(* Logix 5000 project; controller LeakTestAuto vendor 1 type 14 code 226 rev 37.11; software revision 37.01; part 3 of 13 *)
(* tags used below, declared in another part *)
   iarsiInputFromDTE : SINT[496];   // Input array from DTE to PLC
   iiInputStartAdd : INT;   // It is the start of the DTE102:I from which the data has to be read depending upon the channel is being used by the user
   oarsiOutputToDTE : SINT[496];   // Output array from PLC to DTE
   iLoopHandlerVar1 : INT;   // Local tag - Loop Handler variable 1
   iArraySize : INT;
   scDTE102_Handling : DTE102_CmdModule;
   iStateMachine_RWH_CMD : INT;   // Local tag - State machine handling variable for AOI logic
(* RWH_CMD, continued *)

ROUTINE Prescan   (* structured text *)
// Intialisation routine
   	(*Intialise*)
   
   	scDTE102_Handling.ActivateCommand.AO	:= 0;
   	scDTE102_Handling.ActivateCommand.WR	:= 0;
   	scDTE102_Handling.ActivateCommand.RD	:= 0;
   	scDTE102_Handling.ActivateCommand.UR	:= 0;
   	scDTE102_Handling.ActivateCommand.ER	:= 0;
   	scDTE102_Handling.ActivateCommand.DR	:= 0;
   	scDTE102_Handling.ActivateCommand.CM	:= 0;
   	scDTE102_Handling.ActivateCommand.TR	:= (iarsiInputFromDTE[iiInputStartAdd+1].0);
   
   	SIZE(oarsiOutputToDTE,0,iArraySize);
   	FOR iLoopHandlerVar1 :=0 TO iArraySize BY 1 DO;
           oarsiOutputToDTE[iLoopHandlerVar1] := 0;
       END_FOR;
   
   	iStateMachine_RWH_CMD := 25999;
   
END_ROUTINE
END_ADD_ON_INSTRUCTION

ADD_ON_INSTRUCTION SINT_TO_INT   (* revision 1.0 *)
// Converts the negative values of SINT variable to positive values and stores it to a INT variable.
// -128 to -1 = 128 to 255
// 0 to 127 = 0 to 127
// So -128 to 127 to 0 to 255
VAR_INPUT
   iSINT_var : SINT; {required}
END_VAR
VAR_OUTPUT
   oINT_var : INT; {visible}
END_VAR

ROUTINE Logic   (* structured text *)
   IF(iSINT_var<0)THEN
   	oINT_var := 256 + iSINT_var;
   ELSE
   	oINT_var := iSINT_var;
   END_IF;
END_ROUTINE
END_ADD_ON_INSTRUCTION

VAR_GLOBAL   (* controller tags *)
   AOI_IOCounter : AOI_IOCounter;
   ConveyorPurgeCounter : DINT;   // Outfeed Coveyor Purge Counter
   DateString : String20 := '01/14/1998';
   DateTimeString : String20 := '01/14/1998 03:13:45';
   Delay_TMR : TIMER[11] := ([0].PRE := 500, [1].PRE := 500, [3].PRE := 1000, [10].PRE := 100);   // Delay Timers
   HMI_ClearProcessFaultCounts_PB : BOOL;
   HMI_PurgeCycleSP : DINT := 20;   // HMI Purge Cycles Setpoint
   I_OP220_N3_CONVEYOR_CLEAT : ALIAS FOR Local:3:I.Pt13.Data;
   I_OP220_N3_CONVEYOR_LOAD : ALIAS FOR Local:3:I.Pt12.Data;
   I_OP220_N3_CONVEYOR_UNLOAD : ALIAS FOR Local:3:I.Pt14.Data;
   I_OP220_N3_CTS_AIR_OK : ALIAS FOR Local:3:I.Pt08.Data;
   I_OP220_N3_DUT_PRE_NEST_0 : ALIAS FOR Local:3:I.Pt00.Data;
   I_OP220_N3_DUT_PRE_NEST_1 : ALIAS FOR Local:3:I.Pt01.Data;
   I_OP220_N3_DUT_PRE_NEST_2 : ALIAS FOR Local:3:I.Pt02.Data;
   I_OP220_N3_MAIN_AIR_OK : ALIAS FOR Local:3:I.Pt07.Data;
   I_OP220_N3_NEST1_EXTEND : ALIAS FOR Local:3:I.Pt04.Data;
   I_OP220_N3_NEST1_HOME : ALIAS FOR Local:3:I.Pt03.Data;
   I_OP220_N3_NEST2_EXTEND : ALIAS FOR Local:3:I.Pt06.Data;
   I_OP220_N3_NEST2_HOME : ALIAS FOR Local:3:I.Pt05.Data;
   I_OP220_N3_REJECT_BIN_OK : ALIAS FOR Local:3:I.Pt09.Data;
   I_OP220_N3_REJECT_CHUTE_PART : ALIAS FOR Local:3:I.Pt10.Data;
   I_OP220_N4_AC_SURGE_OK : ALIAS FOR Local:4:I.Pt00.Data;
   I_OP220_N4_CONVEYOR_ALARM_OK : ALIAS FOR Local:4:I.Pt03.Data;
   I_OP220_N4_CONVEYOR_SPEED : ALIAS FOR Local:4:I.Pt02.Data;
   I_OP220_N4_DC_OK : ALIAS FOR Local:4:I.Pt01.Data;
   I_OP220_N4_DC_OK_PS2 : ALIAS FOR Local:4:I.Pt04.Data;
   Ignition_Bypass : BOOL := 1;
   Ignition_DataReady : BOOL;
   Ignition_DataReceived : BOOL;
   IOCounterHasRef : BOOL := 1;
   IOCounterLastData : INT[8] := ([0] := 13997, [1] := 27, [2] := -31920);
   IOLabels : STRING[128] := ([0] := 'SI_OP220_N1_LASER_AREA_NC12', [1] := 'SI_OP220_N1_LASER_GUARD_NC12', [3] := 'SI_OP220_N1_SSR_12', [4] := 'SI_OP220_N1_CTRL_VLAVE_NC1', [8] := 'SO_OP220_N2_SSR_1', [9] := 'SO_OP220_N2_SSR_2', [16] := 'I_OP220_N3_DUT_PRE_NEST_0', [17] := 'I_OP220_N3_DUT_PRE_NEST_1', [18] := 'I_OP220_N3_DUT_PRE_NEST_2', [19] := 'I_OP220_N3_NEST1_HOME', [20] := 'I_OP220_N3_NEST1_EXTEND', [21] := 'I_OP220_N3_NEST2_HOME', [22] := 'I_OP220_N3_NEST2_EXTEND', [23] := 'I_OP220_N3_MAIN_AIR_OK', [25] := 'I_OP220_N3_REJECT_BIN_OK', [26] := 'I_OP220_N3_REJECT_CHUTE_PART', [28] := 'I_OP220_N3_CONVEYOR_LOAD', [29] := 'I_OP220_N3_CONVEYOR_CLEAT', [30] := 'I_OP220_N3_CONVEYOR_UNLOAD', [32] := 'I_OP220_N4_AC_SURGE_OK', [33] := 'I_OP220_N4_DC_OK', [34] := 'I_OP220_N4_CONVEYOR_SPEED', [35] := 'I_OP220_N4_CONVEYOR_ALARM_OK', [36] := 'I_OP220_N4_DC_OK_PS2', [48] := 'O_OP220_N5_EN_LT_GN', [49] := 'O_OP220_N5_EN_LT_YE', [50] := 'O_OP220_N5_EN_LT_RD', [51] := 'O_OP220_N5_EN_LT_BU', [52] := 'O_OP220_N5_EN_MAIN_AIR', [53] := 'O_OP220_N5_EN_NEST1_EXT', [54] := 'O_OP220_N5_EN_NEST1_HOME', [55] := 'O_OP220_N5_EN_NEST2_EXT', [56] := 'O_OP220_N5_EN_NEST2_HOME', [57] := 'O_OP220_N5_EN_ROBOT_LATCHOFF', [58] := 'O_OP220_N5_EN_CONV_ALM_RST', [59] := 'O_OP220_N5_CONV_REV', [60] := 'O_OP220_N5_CONV_FWD', [62] := 'O_OP220_N5_EN_GRIPPER_GRIP', [63] := 'O_OP220_N5_EN_GRIPPER_UNGRIP');
   IOResetArray : INT[8];
   IOTriggerCounts : UDINT[128] := ([0] := 204475, [1] := 372996, [2] := 290087, [3] := 284, [4] := 293, [5] := 289, [6] := 294, [7] := 60, [8] := 522, [9] := 268, [10] := 461, [11] := 1169, [12] := 501, [13] := 259, [14] := 218085, [16] := 969915, [17] := 969727, [18] := 63, [19] := 1025, [21] := 84232, [22] := 84239, [23] := 72816, [24] := 72798, [25] := 504, [26] := 4412, [28] := 201969, [29] := 3, [30] := 359118, [31] := 359118);
   James_Dint : DINT := 31;   // James Test Word
   LastPLCEdit : String20 := '01/14/1998 03:11:29';
   LastPLCEditHistory : String20[20] := ([0] := '01/14/1998 03:11:29', [1] := '01/14/1998 02:38:23', [2] := '01/14/1998 02:28:45', [3] := '01/14/1998 02:24:53', [4] := '01/11/1998 11:02:53', [5] := '01/11/1998 10:59:23', [6] := '01/11/1998 10:58:09', [7] := '01/11/1998 10:55:51', [8] := '01/11/1998 05:50:18', [9] := '01/11/1998 05:46:44', [10] := '01/11/1998 05:46:03', [11] := '01/11/1998 05:24:08', [12] := '01/11/1998 05:15:43', [13] := '01/11/1998 04:51:18', [14] := '01/11/1998 04:33:38', [15] := '01/11/1998 03:28:20', [16] := '01/10/1998 12:07:04', [17] := '01/10/1998 12:06:39', [18] := '01/10/1998 12:05:41', [19] := '01/10/1998 11:56:52');
   NoData : AB:5000_DI16:I:0;
   null : STRING;
   O_OP220_N5_CONV_FWD : ALIAS FOR Local:5:O.Pt12.Data;
   O_OP220_N5_CONV_REV : ALIAS FOR Local:5:O.Pt11.Data;
   O_OP220_N5_EN_CONV_ALM_RST : ALIAS FOR Local:5:O.Pt10.Data;
   O_OP220_N5_EN_GRIPPER_GRIP : ALIAS FOR Local:5:O.Pt14.Data;
   O_OP220_N5_EN_GRIPPER_UNGRIP : ALIAS FOR Local:5:O.Pt15.Data;
   O_OP220_N5_EN_LT_BU : ALIAS FOR Local:5:O.Pt03.Data;
   O_OP220_N5_EN_LT_GN : ALIAS FOR Local:5:O.Pt00.Data;
   O_OP220_N5_EN_LT_RD : ALIAS FOR Local:5:O.Pt02.Data;
   O_OP220_N5_EN_LT_YE : ALIAS FOR Local:5:O.Pt01.Data;
   O_OP220_N5_EN_MAIN_AIR : ALIAS FOR Local:5:O.Pt04.Data;
   O_OP220_N5_EN_NEST1_EXT : ALIAS FOR Local:5:O.Pt05.Data;
   O_OP220_N5_EN_NEST1_HOME : ALIAS FOR Local:5:O.Pt06.Data;
   O_OP220_N5_EN_NEST2_EXT : ALIAS FOR Local:5:O.Pt07.Data;
   O_OP220_N5_EN_NEST2_HOME : ALIAS FOR Local:5:O.Pt08.Data;
   O_OP220_N5_EN_ROBOT_LATCHOFF : ALIAS FOR Local:5:O.Pt09.Data;
   Oneshot : DINT;   // Oneshots
   OP220_ConsumedFromMain : DINT[50] := ([0] := 2, [1] := 2);
   OP220_ConsumedFromMain_PurgeModeEn : BOOL;
   OP220_ConsumedFromMain_RobotPickupSafe : BOOL := 1;
   OP220_EStop_OK : BOOL := 1;
   OP220_EStopTest_DCS : DCI_STOP := (ChannelA := 1, ChannelB := 1, InputStatus := 1, RestartType := 1, ColdStartType := 1, DiscrepancyTime := 250, O1 := 1);
   OP220_Power : BOOL := 1;
   OP220_ProducedForMain : DINT[50] := ([0] := 3); {produced}
   PLC : AOI_PLC := (AlwaysOn := 1, FlasherSlow := 1, SlowFlashTime := 2000, MediumFlashTime := 1000, FastFlashTime := 500, Year := 1998, Day := 14, Month := 1, Hour := 3, Minute := 13, Second := 45, MicroSecond := 714855, DOY := 14, SetTimePB := 1);
   Produced_SetTime : udt_Produced_SetTime := (SetTime[0] := 2020, SetTime[1] := 5, SetTime[2] := 21, SetTime[3] := 15, SetTime[4] := 59, SetTime[5] := 15); {produced}
   Purge_Count_DN : BOOL;   // Purge Counter Completed
   ShiftChange : BOOL;
   ShiftNumber : SINT := 2;
   SI_OP220_N1_CTRL_VLAVE_NC1 : ALIAS FOR Local:1:I.Pt04.Data;
   SI_OP220_N1_LASER_AREA_NC12 : ALIAS FOR Local:1:I.Pt00.Data;
   SI_OP220_N1_LASER_GUARD_NC12 : ALIAS FOR Local:1:I.Pt01.Data;
   SI_OP220_N1_SSR_12 : ALIAS FOR Local:1:I.Pt03.Data;
   SO_OP220_N2_SSR_1 : ALIAS FOR Local:2:O.Pt00.Data;
   SO_OP220_N2_SSR_2 : ALIAS FOR Local:2:O.Pt01.Data;
   ST1_Ignition_DataReady : BOOL;
   ST1_Ignition_DataReady_Setup : BOOL;
   ST1_Ignition_DataReceived : BOOL;
   ST1_Ignition_SerialNum : STRING;
   ST1_Ignition_Status : DINT := -10;
   ST2_Ignition_DataReady : BOOL;
   ST2_Ignition_DataReady_Setup : BOOL;
   ST2_Ignition_DataReceived : BOOL;
   ST2_Ignition_SerialNum : STRING;
   ST2_Ignition_Status : DINT := -10;
   TimeString : String20 := '03:13:45';
   TON_PLC_BootUp : TIMER := (PRE := 10000);
END_VAR

PROGRAM MainProgram   (* main routine MainRoutine *)
VAR
   AOI_Barcode_Comms : AOI_CommStatus := (Cmd := 1, stsRunning := 1, stsFaultCode := 272);
   AOI_CapActuators_Seq : AOI_Sequencer_x64 := (inpNextStepInterlock := 1);
   AOI_CapCTS_Seq : AOI_Sequencer_x64 := (inpNextStepInterlock := 1);
   AOI_CapCylinders_Seq : AOI_Sequencer_x64 := (inpNextStepInterlock := 1);
   AOI_CapFail_Seq : AOI_Sequencer_x64 := (inpNextStepInterlock := 1);
   AOI_CapPass_Seq : AOI_Sequencer_x64 := (inpNextStepInterlock := 1);
   AOI_CapRobot_Seq : AOI_Sequencer_x64 := (inpNextStepInterlock := 1);
   AOI_CapShuffle_Seq : AOI_Sequencer_x64 := (inpNextStepInterlock := 1);
   AOI_Conveyor_Seq : AOI_Sequencer_x64 := (inpNextStepInterlock := 1);
   AOI_CTS1 : AOI_CTS_INSTRUMENT := (Change_Program_Number := 3, Current_Program_Number := 3, Instrument_Ready := 1, Program_Accept := 1, Last_Result_Unique_ID := 9525, Last_Result_Channel_Number := 1, Last_Result_Progam_Number := 3, Last_Result_Evaluation_Code := 1, Last_Result_Year := 26, Last_Result_Month := 9, Last_Result_Date := 28, Last_Result_Hour := 11, Last_Result_Minute := 13, Last_Result_Second := 13, UID_of_Desired_Results := 9478, Include_Detailed_Results := 1, Results_Ready := 1, UID_Time := 1300, Ready := 1);
   AOI_CTS1_Comms : AOI_CommStatus := (Cmd := 1, stsRunning := 1, stsFaultCode := 272);
   AOI_CTS1_Seq : AOI_Sequencer_x64 := (inpNextStepInterlock := 1);
   AOI_CTS2 : AOI_CTS_INSTRUMENT := (Change_Program_Number := 3, Current_Program_Number := 3, Instrument_Ready := 1, Program_Accept := 1, Last_Result_Unique_ID := 10924, Last_Result_Channel_Number := 1, Last_Result_Progam_Number := 3, Last_Result_Evaluation_Code := 1, Last_Result_Year := 26, Last_Result_Month := 9, Last_Result_Date := 28, Last_Result_Hour := 11, Last_Result_Second := 7, UID_of_Desired_Results := 10592, Include_Detailed_Results := 1, Results_Ready := 1, UID_Time := 1300, Ready := 1);
   AOI_CTS2_Comms : AOI_CommStatus := (Cmd := 1, stsRunning := 1, stsFaultCode := 272);
   AOI_CTS2_Seq : AOI_Sequencer_x64 := (inpNextStepInterlock := 1);
   AOI_GetShift : AOI_GetShift := (PLCHour := 3, ShiftNumber := 2);
   AOI_OP220_HomingSeq : AOI_Sequencer_x64;
   AOI_OP220_Seq : AOI_Sequencer_x64 := (inpNextStepInterlock := 1);
   AOI_RFID_Comms : AOI_CommStatus := (Cmd := 1, stsRunning := 1, stsFaultCode := 516);
   AOI_RFID_LoadingNest_Comms : AOI_CommStatus := (Cmd := 1, stsRunning := 1, stsFaultCode := 272);
   AOI_Robot_Comms : AOI_CommStatus := (Cmd := 1, stsRunning := 1, stsFaultCode := 272);
   AOI_RobotPos : AOI_RobotPositions := (Barcode := 1, TestingNest1 := 2, TestingNest2 := 3, PassChute := 4, FailChute := 5);
   AOI_SeqSteps : AOI_StandardSeqSteps := (Start := 1000, ResultProcessing := 8000, Complete := 9000);
   AOI_SRX100 : AOI_KeyenceBarcode := (ReadSuccess := 1);
   Barcode_ResultData : STR_Barcode := '260911463C';
   BarcodeBypass : BOOL;
   BarcodeInputs : udt_KeyenceScannerInputs := (READY := 1, ResultDataReadyCount := 25, ResultDataUpdateCount := 25, MasterTriggerCount := 25, ResultDataSize := 10, ResultData[0] := 50, ResultData[1] := 54, ResultData[2] := 48, ResultData[3] := 51, ResultData[4] := 56, ResultData[5] := 48, ResultData[6] := 56, ResultData[7] := 48, ResultData[8] := 57, ResultData[9] := 67);
   BarcodeOutputs : udt_KeyenceScannerOutputs;
   BarcodeScanner : udt_OutputStructure := (IL := 1);
   CapActuators_BarcodeBad : COUNTER := (PRE := 999999999, CU := 1);
   CapActuators_BarcodeGood : COUNTER := (PRE := 999999999, ACC := 111, CU := 1);
   CapActuators_CTS1Bad : COUNTER := (PRE := 999999999, CU := 1);
   CapActuators_CTS1Good : COUNTER := (PRE := 999999999, ACC := 10, CU := 1);
   CapActuators_CTS2Bad : COUNTER := (PRE := 999999999, CU := 1);
   CapActuators_CTS2Good : COUNTER := (PRE := 999999999, ACC := 3, CU := 1);
   CapActuators_Nest1HasPart : BOOL := 1;
   CapActuators_Nest2HasPart : BOOL;
   CapActuators_Seq : udt_SequenceStructure_X64 := (ONS := -7937, CurrentCycleTime := 409000.0, StepTimer.PRE := 999999999, CycleTimer.PRE := 999999999);
   CapCTS_CTS1Bad : COUNTER := (PRE := 999999999, ACC := 356, CU := 1);
   CapCTS_CTS1Good : COUNTER := (PRE := 999999999, ACC := 2730, CU := 1);
   CapCTS_CTS2Bad : COUNTER := (PRE := 999999999, ACC := 1, CU := 1);
   CapCTS_CTS2Good : COUNTER := (PRE := 999999999, ACC := 3085, CU := 1);
   CapCTS_Nest1HasPart : BOOL := 1;
   CapCTS_Nest2HasPart : BOOL := 1;
   CapCTS_Seq : udt_SequenceStructure_X64 := (ONS := -8132, StepHistory[0] := 2000, StepHistory[1] := 2010, StepHistory[2] := 2000, StepHistory[3] := 2010, StepHistory[4] := 2000, StepHistory[5] := 2010, StepHistory[6] := 2000, StepHistory[7] := 2010, StepHistory[8] := 2000, StepHistory[9] := 2010, StepHistory[10] := 2000, StepHistory[11] := 2010, StepHistory[12] := 2000, StepHistory[13] := 2010, StepHistory[14] := 2000, StepHistory[15] := 2010, StepHistory[16] := 2000, StepHistory[17] := 2010, StepHistory[18] := 2000, StepHistory[19] := 2010, StepHistory[20] := 2000, StepHistory[21] := 2010, StepHistory[22] := 2000, StepHistory[23] := 2010, StepHistory[24] := 2000, StepHistory[25] := 2010, StepHistory[26] := 2000, StepHistory[27] := 2010, StepHistory[28] := 2000, StepHistory[29] := 2010, StepHistory[30] := 2000, StepHistory[31] := 2010, StepHistory[32] := 2000, StepHistory[33] := 2010, StepHistory[34] := 2000, StepHistory[35] := 2010, StepHistory[36] := 2000, StepHistory[37] := 2010, StepHistory[38] := 2000, StepHistory[39] := 2010, StepHistory[40] := 2000, StepHistory[41] := 2010, StepHistory[42] := 2000, StepHistory[43] := 2010, StepHistory[44] := 2000, StepHistory[45] := 2010, StepHistory[46] := 2000, StepHistory[47] := 2010, StepHistory[48] := 2000, StepHistory[49] := 2010, StepHistory[50] := 2000, StepHistory[51] := 2010, StepHistory[52] := 2000, StepHistory[53] := 2010, StepHistory[54] := 2000, StepHistory[55] := 2010, StepHistory[56] := 2000, StepHistory[57] := 2010, StepHistory[58] := 2000,
        StepHistory[59] := 2010, StepHistory[60] := 2000, StepHistory[61] := 2010, StepHistory[62] := 2000, StepHistory[63] := 2010, CurrentCycleTime := 66060.766, CurrentStepCycleTime := 387.139, StepTimeHistory[0] := 0.035, StepTimeHistory[1] := 21.3, StepTimeHistory[2] := 0.04, StepTimeHistory[3] := 21.295, StepTimeHistory[4] := 0.035, StepTimeHistory[5] := 21.266, StepTimeHistory[6] := 0.034, StepTimeHistory[7] := 21.271, StepTimeHistory[8] := 0.033, StepTimeHistory[9] := 21.285, StepTimeHistory[10] := 0.041, StepTimeHistory[11] := 21.294, StepTimeHistory[12] := 0.052, StepTimeHistory[13] := 21.304, StepTimeHistory[14] := 0.035, StepTimeHistory[15] := 21.297, StepTimeHistory[16] := 0.036, StepTimeHistory[17] := 21.266, StepTimeHistory[18] := 0.039, StepTimeHistory[19] := 21.292, StepTimeHistory[20] := 0.04, StepTimeHistory[21] := 21.273, StepTimeHistory[22] := 0.035, StepTimeHistory[23] := 21.271, StepTimeHistory[24] := 0.051, StepTimeHistory[25] := 21.29, StepTimeHistory[26] := 0.036, StepTimeHistory[27] := 21.274, StepTimeHistory[28] := 0.041, StepTimeHistory[29] := 21.289, StepTimeHistory[30] := 0.036, StepTimeHistory[31] := 21.285, StepTimeHistory[32] := 0.039, StepTimeHistory[33] := 21.296, StepTimeHistory[34] := 0.05, StepTimeHistory[35] := 21.273, StepTimeHistory[36] := 0.057, StepTimeHistory[37] := 21.274, StepTimeHistory[38] := 0.034, StepTimeHistory[39] := 21.285, StepTimeHistory[40] := 0.05, StepTimeHistory[41] := 21.27, StepTimeHistory[42] := 0.036, StepTimeHistory[43] := 21.29, StepTimeHistory[44] := 0.035, StepTimeHistory[45] := 21.309, StepTimeHistory[46] := 0.051, StepTimeHistory[47] := 21.274, StepTimeHistory[48] := 0.037, StepTimeHistory[49] := 21.315, StepTimeHistory[50] := 0.044, StepTimeHistory[51] := 21.296, StepTimeHistory[52] := 0.035,
        StepTimeHistory[53] := 21.271, StepTimeHistory[54] := 0.034, StepTimeHistory[55] := 21.289, StepTimeHistory[56] := 0.045, StepTimeHistory[57] := 21.29, StepTimeHistory[58] := 0.034, StepTimeHistory[59] := 21.296, StepTimeHistory[60] := 0.035, StepTimeHistory[61] := 21.293, StepTimeHistory[62] := 0.069, StepTimeHistory[63] := 21.691, StepTimer.PRE := 999999999, CycleTimer.PRE := 999999999);
   CapCylinders_Seq : udt_SequenceStructure_X64 := (ONS := -8192);
   CapFail_Seq : udt_SequenceStructure_X64 := (ONS := -8192);
   CapPass_Seq : udt_SequenceStructure_X64 := (ONS := -8191);
   CapRobot_IsNest : BOOL;
   CapRobot_Seq : udt_SequenceStructure_X64 := (ONS := -8191, StepHistory[0] := 2040, StepHistory[1] := 2050, StepHistory[2] := 2060, StepHistory[3] := 2070, StepHistory[4] := 2000, StepHistory[5] := 2010, StepHistory[6] := 2020, StepHistory[7] := 2030, StepHistory[8] := 2050, StepHistory[9] := 2060, StepHistory[10] := 2070, StepHistory[11] := 2000, StepHistory[12] := 2010, StepHistory[13] := 2020, StepHistory[14] := 2030, StepHistory[15] := 2050, StepHistory[16] := 2060, StepHistory[17] := 2070, StepHistory[18] := 2000, StepHistory[19] := 2010, StepHistory[20] := 2020, StepHistory[21] := 2030, StepHistory[22] := 2040, StepHistory[23] := 2050, StepHistory[24] := 2060, StepHistory[25] := 2070, StepHistory[26] := 2000, StepHistory[27] := 2010, StepHistory[28] := 2020, StepHistory[29] := 2030, StepHistory[30] := 2040, StepHistory[31] := 2050, StepHistory[32] := 2060, StepHistory[33] := 2070, StepHistory[34] := 2000, StepHistory[35] := 2010, StepHistory[36] := 2020, StepHistory[37] := 2030, StepHistory[38] := 2050, StepHistory[39] := 2060, StepHistory[40] := 2070, StepHistory[41] := 2000, StepHistory[42] := 2010, StepHistory[43] := 2020, StepHistory[45] := 1000, StepHistory[46] := 2000, StepHistory[47] := 2010, StepHistory[48] := 2020, StepHistory[49] := 2030, StepHistory[50] := 2050, StepHistory[51] := 2060, StepHistory[52] := 2070, StepHistory[53] := 2000, StepHistory[54] := 2010, StepHistory[55] := 2020, StepHistory[56] := 2030, StepHistory[57] := 2040, StepHistory[58] := 2050, StepHistory[59] := 2060,
        StepHistory[60] := 2070, StepHistory[61] := 2000, StepHistory[62] := 2010, StepHistory[63] := 2020, CurrentCycleTime := 15.469, CurrentStepCycleTime := 4.281, StepTimeHistory[0] := 0.099, StepTimeHistory[1] := 0.039, StepTimeHistory[2] := 1.559, StepTimeHistory[3] := 1.559, StepTimeHistory[4] := 1.559, StepTimeHistory[5] := 0.097, StepTimeHistory[6] := 0.029, StepTimeHistory[7] := 1.398, StepTimeHistory[8] := 0.038, StepTimeHistory[9] := 1.468, StepTimeHistory[10] := 1.468, StepTimeHistory[11] := 1.468, StepTimeHistory[12] := 0.088, StepTimeHistory[13] := 0.028, StepTimeHistory[14] := 1.279, StepTimeHistory[15] := 0.039, StepTimeHistory[16] := 1.399, StepTimeHistory[17] := 1.399, StepTimeHistory[18] := 0.028, StepTimeHistory[19] := 0.769, StepTimeHistory[20] := 0.029, StepTimeHistory[21] := 0.758, StepTimeHistory[22] := 0.009, StepTimeHistory[23] := 0.039, StepTimeHistory[24] := 0.66, StepTimeHistory[25] := 0.66, StepTimeHistory[26] := 0.66, StepTimeHistory[27] := 0.66, StepTimeHistory[28] := 0.037, StepTimeHistory[29] := 1.209, StepTimeHistory[30] := 0.099, StepTimeHistory[31] := 0.028, StepTimeHistory[32] := 1.049, StepTimeHistory[33] := 1.049, StepTimeHistory[34] := 1.049, StepTimeHistory[35] := 1.049, StepTimeHistory[36] := 0.036, StepTimeHistory[37] := 0.898, StepTimeHistory[38] := 0.038, StepTimeHistory[39] := 0.849, StepTimeHistory[40] := 0.849, StepTimeHistory[41] := 0.849, StepTimeHistory[42] := 0.849, StepTimeHistory[43] := 0.026, StepTimeHistory[44] := 0.264, StepTimeHistory[45] := 0.264, StepTimeHistory[46] := 0.066, StepTimeHistory[47] := 1.64, StepTimeHistory[48] := 0.059, StepTimeHistory[49] := 1.569, StepTimeHistory[50] := 0.049, StepTimeHistory[51] := 1.65, StepTimeHistory[52] := 1.65, StepTimeHistory[53] := 1.65,
        StepTimeHistory[54] := 0.078, StepTimeHistory[55] := 0.058, StepTimeHistory[56] := 2.87, StepTimeHistory[57] := 0.069, StepTimeHistory[58] := 0.07, StepTimeHistory[59] := 2.87, StepTimeHistory[60] := 2.87, StepTimeHistory[61] := 2.87, StepTimeHistory[62] := 0.067, StepTimeHistory[63] := 0.06, StepTimer.PRE := 999999999, CycleTimer.PRE := 999999999);
   CapRobot_StartPos : DINT;
   CapRobot_TargetPos : DINT := 3;
   CapShuffle_CTS1Bad : COUNTER := (PRE := 999999999, ACC := 2, CU := 1);
   CapShuffle_CTS1Good : COUNTER := (PRE := 999999999, CU := 1);
   CapShuffle_CTS2Bad : COUNTER := (PRE := 999999999, CU := 1);
   CapShuffle_CTS2Good : COUNTER := (PRE := 999999999, ACC := 1, CU := 1);
   CapShuffle_Seq : udt_SequenceStructure_X64 := (ONS := -8161, StepHistory[0] := 5610, StepHistory[1] := 5620, StepHistory[2] := 5630, StepHistory[3] := 5640, StepHistory[4] := 5650, StepHistory[5] := 4000, StepHistory[6] := 4010, StepHistory[9] := 1000, StepHistory[10] := 3000, StepHistory[11] := 3010, StepHistory[12] := 3020, StepHistory[15] := 1000, StepHistory[16] := 3000, StepHistory[17] := 3010, StepHistory[18] := 3020, StepHistory[20] := 1000, StepHistory[21] := 3000, StepHistory[22] := 3010, StepHistory[23] := 3020, StepHistory[25] := 1000, StepHistory[26] := 3000, StepHistory[27] := 3010, StepHistory[28] := 3020, StepHistory[29] := 3030, StepHistory[30] := 3020, StepHistory[31] := 3020, StepHistory[32] := 3010, StepHistory[33] := 3030, StepHistory[34] := 3040, StepHistory[35] := 3050, StepHistory[36] := 3060, StepHistory[37] := 3070, StepHistory[38] := 4000, StepHistory[39] := 4010, StepHistory[40] := 4020, StepHistory[41] := 4030, StepHistory[42] := 5000, StepHistory[43] := 5100, StepHistory[44] := 5110, StepHistory[45] := 5120, StepHistory[46] := 5130, StepHistory[47] := 5400, StepHistory[48] := 5410, StepHistory[49] := 5420, StepHistory[50] := 5430, StepHistory[51] := 5440, StepHistory[52] := 5450, StepHistory[53] := 4000, StepHistory[54] := 4010, StepHistory[55] := 4020, StepHistory[56] := 5000, StepHistory[57] := 5600, StepHistory[58] := 5610, StepHistory[59] := 5620, StepHistory[60] := 5630, StepHistory[61] := 5640, StepHistory[62] := 5650, StepHistory[63] := 4000, CurrentCycleTime := 255.519,
        CurrentStepCycleTime := 42.404, StepTimeHistory[0] := 0.879, StepTimeHistory[1] := 0.039, StepTimeHistory[2] := 1.569, StepTimeHistory[3] := 0.029, StepTimeHistory[4] := 1.059, StepTimeHistory[5] := 1.059, StepTimeHistory[6] := 1.059, StepTimeHistory[7] := 4.506, StepTimeHistory[8] := 96.458, StepTimeHistory[9] := 19.876, StepTimeHistory[10] := 0.051, StepTimeHistory[11] := 1.66, StepTimeHistory[12] := 0.06, StepTimeHistory[13] := 0.728, StepTimeHistory[14] := 0.728, StepTimeHistory[15] := 0.728, StepTimeHistory[16] := 0.102, StepTimeHistory[17] := 1.639, StepTimeHistory[18] := 0.059, StepTimeHistory[19] := 13.077, StepTimeHistory[20] := 13.077, StepTimeHistory[21] := 0.07, StepTimeHistory[22] := 1.638, StepTimeHistory[23] := 0.059, StepTimeHistory[24] := 33.884, StepTimeHistory[25] := 33.884, StepTimeHistory[26] := 0.058, StepTimeHistory[27] := 1.648, StepTimeHistory[28] := 0.069, StepTimeHistory[29] := 57.197, StepTimeHistory[30] := 57.197, StepTimeHistory[31] := 10.171, StepTimeHistory[32] := 12.984, StepTimeHistory[33] := 66.124, StepTimeHistory[34] := 0.059, StepTimeHistory[35] := 3.51, StepTimeHistory[36] := 0.059, StepTimeHistory[37] := 3.429, StepTimeHistory[38] := 5.691, StepTimeHistory[39] := 0.551, StepTimeHistory[40] := 5.877, StepTimeHistory[41] := 0.545, StepTimeHistory[42] := 0.545, StepTimeHistory[43] := 0.06, StepTimeHistory[44] := 1.879, StepTimeHistory[45] := 0.059, StepTimeHistory[46] := 10.247, StepTimeHistory[47] := 0.071, StepTimeHistory[48] := 4.469, StepTimeHistory[49] := 0.059, StepTimeHistory[50] := 4.719, StepTimeHistory[51] := 0.069, StepTimeHistory[52] := 1.799, StepTimeHistory[53] := 5.676, StepTimeHistory[54] := 0.548, StepTimeHistory[55] := 0.548, StepTimeHistory[56] := 0.548, StepTimeHistory[57] := 0.061, StepTimeHistory[58] := 1.649,
        StepTimeHistory[59] := 0.099, StepTimeHistory[60] := 4.49, StepTimeHistory[61] := 0.059, StepTimeHistory[62] := 3.418, StepTimeHistory[63] := 5.671, StepTimer.PRE := 999999999, CycleTimer.PRE := 999999999);
   Config_ConveyorHomeCounter : DINT;
   Config_ConveyorHomeCounterEnter : BOOL;
   Config_CylinderWaitTime : DINT := 500;
   Config_CylinderWaitTimeEnter : BOOL;
   Config_MaxFailCount : DINT := 10;
   Config_MaxFailCountEnter : BOOL;
   Conveyor : udt_OutputStructure := (CMD := 1);
   Conveyor_Seq : udt_SequenceStructure_X64 := (StepHistory[0] := 1010, StepHistory[1] := 9000, StepHistory[3] := 1000, StepHistory[4] := 1010, StepHistory[5] := 9000, StepHistory[7] := 1000, StepHistory[8] := 1010, StepHistory[9] := 9000, StepHistory[10] := 1000, StepHistory[11] := 1010, StepHistory[12] := 9000, StepHistory[14] := 1000, StepHistory[15] := 1010, StepHistory[16] := 9000, StepHistory[18] := 1000, StepHistory[19] := 1010, StepHistory[20] := 9000, StepHistory[21] := 1000, StepHistory[22] := 1010, StepHistory[23] := 9000, StepHistory[24] := 1000, StepHistory[25] := 1010, StepHistory[26] := 9000, StepHistory[27] := 1000, StepHistory[28] := 1010, StepHistory[29] := 9000, StepHistory[30] := 1000, StepHistory[31] := 1010, StepHistory[32] := 9000, StepHistory[33] := 1000, StepHistory[34] := 1010, StepHistory[35] := 9000, StepHistory[36] := 1000, StepHistory[37] := 1010, StepHistory[38] := 9000, StepHistory[39] := 1000, StepHistory[40] := 1010, StepHistory[41] := 9000, StepHistory[42] := 1000, StepHistory[43] := 1010, StepHistory[44] := 9000, StepHistory[45] := 1000, StepHistory[46] := 1010, StepHistory[47] := 9000, StepHistory[48] := 1000, StepHistory[49] := 1010, StepHistory[50] := 9000, StepHistory[51] := 1000, StepHistory[52] := 1010, StepHistory[53] := 9000, StepHistory[54] := 1000, StepHistory[55] := 1010, StepHistory[56] := 9000, StepHistory[58] := 1000, StepHistory[59] := 1010, StepHistory[60] := 9000, StepHistory[61] := 1000, StepHistory[62] := 1010, StepHistory[63] := 9000, StepDescriptionPointer := -30912,
        AverageCycleTime := 2.2289, PreviousCycleTime := 2706.0, CycleTimeHistory[0] := 2.488, CycleTimeHistory[1] := 2.453, CycleTimeHistory[2] := 2.542, CycleTimeHistory[3] := 2.472, CycleTimeHistory[4] := 2.482, CycleTimeHistory[5] := 2.503, CycleTimeHistory[6] := 2.524, CycleTimeHistory[7] := 2.365, CycleTimeHistory[8] := 2.46, CurrentStepCycleTime := 2.323, StepTimeHistory[0] := 2.299, StepTimeHistory[1] := 2.299, StepTimeHistory[2] := 2.299, StepTimeHistory[3] := 0.12, StepTimeHistory[4] := 2.424, StepTimeHistory[5] := 2.424, StepTimeHistory[6] := 2.424, StepTimeHistory[7] := 0.123, StepTimeHistory[8] := 2.219, StepTimeHistory[9] := 2.219, StepTimeHistory[10] := 0.125, StepTimeHistory[11] := 2.353, StepTimeHistory[12] := 2.353, StepTimeHistory[13] := 2.353, StepTimeHistory[14] := 0.126, StepTimeHistory[15] := 2.303, StepTimeHistory[16] := 2.303, StepTimeHistory[17] := 2.303, StepTimeHistory[18] := 0.125, StepTimeHistory[19] := 2.343, StepTimeHistory[20] := 2.343, StepTimeHistory[21] := 0.13, StepTimeHistory[22] := 2.363, StepTimeHistory[23] := 2.363, StepTimeHistory[24] := 0.133, StepTimeHistory[25] := 2.314, StepTimeHistory[26] := 2.314, StepTimeHistory[27] := 0.128, StepTimeHistory[28] := 2.343, StepTimeHistory[29] := 2.343, StepTimeHistory[30] := 0.129, StepTimeHistory[31] := 2.338, StepTimeHistory[32] := 2.338, StepTimeHistory[33] := 0.133, StepTimeHistory[34] := 2.34, StepTimeHistory[35] := 2.34, StepTimeHistory[36] := 0.123, StepTimeHistory[37] := 2.364, StepTimeHistory[38] := 2.364, StepTimeHistory[39] := 0.127, StepTimeHistory[40] := 2.323, StepTimeHistory[41] := 2.323, StepTimeHistory[42] := 0.131, StepTimeHistory[43] := 2.41, StepTimeHistory[44] := 2.41, StepTimeHistory[45] := 0.117, StepTimeHistory[46] := 2.353, StepTimeHistory[47] := 2.353,
        StepTimeHistory[48] := 0.121, StepTimeHistory[49] := 2.36, StepTimeHistory[50] := 2.36, StepTimeHistory[51] := 0.137, StepTimeHistory[52] := 2.364, StepTimeHistory[53] := 2.364, StepTimeHistory[54] := 0.132, StepTimeHistory[55] := 2.39, StepTimeHistory[56] := 2.39, StepTimeHistory[57] := 2.39, StepTimeHistory[58] := 0.129, StepTimeHistory[59] := 2.234, StepTimeHistory[60] := 2.234, StepTimeHistory[61] := 0.135, StepTimeHistory[62] := 2.323, StepTimeHistory[63] := 2.323, StepTimer.PRE := 999999999, CycleTimer.PRE := 999999999);
   ConveyorCleatSensorFault : BOOL;
   ConveyorHasParts : BOOL;
   ConveyorHomeCounter : COUNTER := (DN := 1);
   CTS1_BarcodeWrite : STRING80;
   CTS1_BasicResult : MESSAGE;
        MessageParameters(ServiceCode := 16#000e, DestinationTag := CTS1_Result.Basic, ...)
   CTS1_DataRead : STRING80;
   CTS1_DetailResult : MESSAGE;
        MessageParameters(ServiceCode := 16#000e, DestinationTag := CTS1_Result.Detailed, ...)
   CTS1_Inputs : udt_CTS_INPUTS_FROM := (Discrete_Status_Data := -16384, Active_program_num := 3, unique_id := 9525, channel_num := 1, program_num := 3, sequence_num := 3, seq_unique_ID := 9525, evaluation_code := 1, year := 26, month := 9, date := 28, hour := 11, minutes := 13, seconds := 13, flags := 16, test_type := 131, Measurement_data[0].Variable_code := 164, Measurement_data[0].Unit_code := 167, Measurement_data[0].result_measurement := 1.0, Measurement_data[1].Variable_code := 164, Measurement_data[1].Unit_code := 167, Measurement_data[1].result_measurement := 2.0);
   CTS1_LastResultEval : STRING16;
   CTS1_LastTestUID : DINT := 9478;
   CTS1_NextTestUID : DINT := 9478;
   CTS1_NumTestsInSeq : SINT := 2;
   CTS1_Outputs : udt_CTS_OUTPUTS_TO := (program_num := 3);
   CTS1_ReadMsg : MESSAGE;
        MessageParameters(ServiceCode := 16#000e, DestinationTag := CTS1_DataRead.DATA[0], ...)
   CTS1_Ready : DINT;
   CTS1_Result : udt_CTS_RESULT := (UID := 9478, Basic.unique_id := 9478, Basic.channel_num := 1, Basic.program_num := 2, Basic.evaluation_code := 1, Basic.test_port := 1, Basic.year := 26, Basic.month := 9, Basic.date := 24, Basic.hour := 19, Basic.minute := 52, Basic.second := 10, Basic.flags := 12, Basic.Num_tests := 1, Basic.test_elements.test_type := 66, Basic.test_elements.test_eval := 1, Basic.test_elements.num_elements := 16, Detailed.unique_id := 9478, Detailed.num_elements := 16, Detailed.Test_Type := 66, Detailed.element_data[0].Variable_code := 61, Detailed.element_data[0].prec_code := 2, Detailed.element_data[0].Unit_code := 60, Detailed.element_data[0].result_measurement := -0.051409006, Detailed.element_data[1].Variable_code := 28, Detailed.element_data[1].prec_code := 3, Detailed.element_data[1].Unit_code := 41, Detailed.element_data[1].result_measurement := 0.00056345016, Detailed.element_data[2].Variable_code := 13, Detailed.element_data[2].prec_code := 3, Detailed.element_data[2].Unit_code := 12, Detailed.element_data[2].result_measurement := 5.0597124, Detailed.element_data[3].Variable_code := 75, Detailed.element_data[3].prec_code := 2, Detailed.element_data[3].Unit_code := 60, Detailed.element_data[4].Variable_code := 60, Detailed.element_data[4].prec_code := 2, Detailed.element_data[4].Unit_code := 60, Detailed.element_data[4].result_measurement := -0.08158386, Detailed.element_data[5].Variable_code := 56, Detailed.element_data[5].prec_code := 3, Detailed.element_data[5].Unit_code := 41, Detailed.element_data[5].result_measurement := 9.778887e-05, Detailed.element_data[6].Variable_code := 55, Detailed.element_data[6].prec_code := 3, Detailed.element_data[6].Unit_code := 12, Detailed.element_data[6].result_measurement := 5.0597124, Detailed.element_data[7].Variable_code := 58, Detailed.element_data[7].prec_code := 2, Detailed.element_data[7].Unit_code := 60, Detailed.element_data[7].result_measurement := -1.0002404, Detailed.element_data[8].Variable_code := 59, Detailed.element_data[8].prec_code := 2, Detailed.element_data[8].Unit_code := 60, Detailed.element_data[8].result_measurement := 1.0002404, Detailed.element_data[9].Variable_code := 12, Detailed.element_data[9].prec_code := 3, Detailed.element_data[9].Unit_code := 12, Detailed.element_data[9].result_measurement := 5.000001, Detailed.element_data[10].Variable_code := 62,
        Detailed.element_data[10].prec_code := 2, Detailed.element_data[10].Unit_code := 60, Detailed.element_data[10].result_measurement := 1.0902061, Detailed.element_data[11].Variable_code := 21, Detailed.element_data[11].prec_code := 3, Detailed.element_data[11].Unit_code := 41, Detailed.element_data[11].result_measurement := 0.0015180558, Detailed.element_data[12].Variable_code := 25, Detailed.element_data[12].prec_code := 3, Detailed.element_data[12].Unit_code := 41, Detailed.element_data[12].result_measurement := 0.021727756, Detailed.element_data[13].Variable_code := 216, Detailed.element_data[13].prec_code := 3, Detailed.element_data[13].Unit_code := 41, Detailed.element_data[13].result_measurement := 0.00085681677, Detailed.element_data[14].Variable_code := 218, Detailed.element_data[14].prec_code := 3, Detailed.element_data[14].Unit_code := 41, Detailed.element_data[14].result_measurement := 0.01094304, Detailed.element_data[15].Variable_code := 295, Detailed.element_data[15].prec_code := 3, Detailed.element_data[15].Unit_code := 12, Detailed.element_data[15].result_measurement := 5.063093);
   CTS1_ResultHistoryLeak : udt_CTS_RESULT[10] := ([0].UID := 42959, [0].Basic.unique_id := 42959, [0].Basic.channel_num := 1, [0].Basic.program_num := 2, [0].Basic.evaluation_code := 1, [0].Basic.test_port := 1, [0].Basic.year := 26, [0].Basic.month := 6, [0].Basic.date := 4, [0].Basic.hour := 15, [0].Basic.minute := 8, [0].Basic.second := 17, [0].Basic.flags := 12, [0].Basic.Num_tests := 1, [0].Basic.test_elements.test_type := 66, [0].Basic.test_elements.test_eval := 1, [0].Basic.test_elements.num_elements := 16, [0].Detailed.unique_id := 42959, [0].Detailed.num_elements := 16, [0].Detailed.Test_Type := 66, [0].Detailed.element_data[0].Variable_code := 61, [0].Detailed.element_data[0].prec_code := 2, [0].Detailed.element_data[0].Unit_code := 60, [0].Detailed.element_data[1].Variable_code := 28, [0].Detailed.element_data[1].prec_code := 3, [0].Detailed.element_data[1].Unit_code := 41, [0].Detailed.element_data[1].result_measurement := -4.656613e-06, [0].Detailed.element_data[2].Variable_code := 13, [0].Detailed.element_data[2].prec_code := 3, [0].Detailed.element_data[2].Unit_code := 12, [0].Detailed.element_data[2].result_measurement := 5.2301817, [0].Detailed.element_data[3].Variable_code := 75, [0].Detailed.element_data[3].prec_code := 2, [0].Detailed.element_data[3].Unit_code := 60, [0].Detailed.element_data[4].Variable_code := 60, [0].Detailed.element_data[4].prec_code := 2, [0].Detailed.element_data[4].Unit_code := 60, [0].Detailed.element_data[4].result_measurement := 0.0027939677, [0].Detailed.element_data[5].Variable_code := 56, [0].Detailed.element_data[5].prec_code := 3, [0].Detailed.element_data[5].Unit_code := 41, [0].Detailed.element_data[5].result_measurement := -4.656613e-06, [0].Detailed.element_data[6].Variable_code := 55, [0].Detailed.element_data[6].prec_code := 3, [0].Detailed.element_data[6].Unit_code := 12, [0].Detailed.element_data[6].result_measurement := 5.2301817, [0].Detailed.element_data[7].Variable_code := 58, [0].Detailed.element_data[7].prec_code := 2, [0].Detailed.element_data[7].Unit_code := 60, [0].Detailed.element_data[7].result_measurement := -1.0002404, [0].Detailed.element_data[8].Variable_code := 59, [0].Detailed.element_data[8].prec_code := 2, [0].Detailed.element_data[8].Unit_code := 60, [0].Detailed.element_data[8].result_measurement := 1.0002404, [0].Detailed.element_data[9].Variable_code := 12, [0].Detailed.element_data[9].prec_code := 3, [0].Detailed.element_data[9].Unit_code := 12, [0].Detailed.element_data[9].result_measurement := 5.000001, [0].Detailed.element_data[10].Variable_code := 62, [0].Detailed.element_data[10].prec_code := 2,
        [0].Detailed.element_data[10].Unit_code := 60, [0].Detailed.element_data[10].result_measurement := 1.1298805, [0].Detailed.element_data[11].Variable_code := 21, [0].Detailed.element_data[11].prec_code := 3, [0].Detailed.element_data[11].Unit_code := 41, [0].Detailed.element_data[11].result_measurement := 4.656613e-06, [0].Detailed.element_data[12].Variable_code := 25, [0].Detailed.element_data[12].prec_code := 3, [0].Detailed.element_data[12].Unit_code := 41, [0].Detailed.element_data[12].result_measurement := 0.023245811, [0].Detailed.element_data[13].Variable_code := 216, [0].Detailed.element_data[13].prec_code := 3, [0].Detailed.element_data[13].Unit_code := 41, [0].Detailed.element_data[13].result_measurement := -3.7252903e-05, [0].Detailed.element_data[14].Variable_code := 218, [0].Detailed.element_data[14].prec_code := 3, [0].Detailed.element_data[14].Unit_code := 41, [0].Detailed.element_data[14].result_measurement := 0.011632219, [0].Detailed.element_data[15].Variable_code := 295, [0].Detailed.element_data[15].prec_code := 3, [0].Detailed.element_data[15].Unit_code := 12, [0].Detailed.element_data[15].result_measurement := 5.23197, [1].UID := 42962, [1].Basic.unique_id := 42962, [1].Basic.channel_num := 1, [1].Basic.program_num := 2, [1].Basic.evaluation_code := 1, [1].Basic.test_port := 1, [1].Basic.year := 26, [1].Basic.month := 6, [1].Basic.date := 4, [1].Basic.hour := 15, [1].Basic.minute := 9, [1].Basic.second := 47, [1].Basic.flags := 12, [1].Basic.Num_tests := 1, [1].Basic.test_elements.test_type := 66, [1].Basic.test_elements.test_eval := 1, [1].Basic.test_elements.num_elements := 16, [1].Detailed.unique_id := 42962, [1].Detailed.num_elements := 16, [1].Detailed.Test_Type := 66, [1].Detailed.element_data[0].Variable_code := 61, [1].Detailed.element_data[0].prec_code := 2, [1].Detailed.element_data[0].Unit_code := 60, [1].Detailed.element_data[0].result_measurement := 0.022351742, [1].Detailed.element_data[1].Variable_code := 28, [1].Detailed.element_data[1].prec_code := 3, [1].Detailed.element_data[1].Unit_code := 41, [1].Detailed.element_data[1].result_measurement := 0.0004656613, [1].Detailed.element_data[2].Variable_code := 13, [1].Detailed.element_data[2].prec_code := 3, [1].Detailed.element_data[2].Unit_code := 12, [1].Detailed.element_data[2].result_measurement := 5.2300653, [1].Detailed.element_data[3].Variable_code := 75, [1].Detailed.element_data[3].prec_code := 2, [1].Detailed.element_data[3].Unit_code := 60, [1].Detailed.element_data[4].Variable_code := 60, [1].Detailed.element_data[4].prec_code := 2, [1].Detailed.element_data[4].Unit_code := 60,
        [1].Detailed.element_data[4].result_measurement := 0.022910535, [1].Detailed.element_data[5].Variable_code := 56, [1].Detailed.element_data[5].prec_code := 3, [1].Detailed.element_data[5].Unit_code := 41, [1].Detailed.element_data[5].result_measurement := 0.00020023435, [1].Detailed.element_data[6].Variable_code := 55, [1].Detailed.element_data[6].prec_code := 3, [1].Detailed.element_data[6].Unit_code := 12, [1].Detailed.element_data[6].result_measurement := 5.2300653, [1].Detailed.element_data[7].Variable_code := 58, [1].Detailed.element_data[7].prec_code := 2, [1].Detailed.element_data[7].Unit_code := 60, [1].Detailed.element_data[7].result_measurement := -1.0002404, [1].Detailed.element_data[8].Variable_code := 59, [1].Detailed.element_data[8].prec_code := 2, [1].Detailed.element_data[8].Unit_code := 60, [1].Detailed.element_data[8].result_measurement := 1.0002404, [1].Detailed.element_data[9].Variable_code := 12, [1].Detailed.element_data[9].prec_code := 3, [1].Detailed.element_data[9].Unit_code := 12, [1].Detailed.element_data[9].result_measurement := 5.000001, [1].Detailed.element_data[10].Variable_code := 62, [1].Detailed.element_data[10].prec_code := 2, [1].Detailed.element_data[10].Unit_code := 60, [1].Detailed.element_data[10].result_measurement := 1.1298805, [1].Detailed.element_data[11].Variable_code := 21, [1].Detailed.element_data[11].prec_code := 3, [1].Detailed.element_data[11].Unit_code := 41, [1].Detailed.element_data[11].result_measurement := 4.656613e-06, [1].Detailed.element_data[12].Variable_code := 25, [1].Detailed.element_data[12].prec_code := 3, [1].Detailed.element_data[12].Unit_code := 41, [1].Detailed.element_data[12].result_measurement := 0.023245811, [1].Detailed.element_data[13].Variable_code := 216, [1].Detailed.element_data[13].prec_code := 3, [1].Detailed.element_data[13].Unit_code := 41, [1].Detailed.element_data[13].result_measurement := -3.7252903e-05, [1].Detailed.element_data[14].Variable_code := 218, [1].Detailed.element_data[14].prec_code := 3, [1].Detailed.element_data[14].Unit_code := 41, [1].Detailed.element_data[14].result_measurement := 0.011632219, [1].Detailed.element_data[15].Variable_code := 295, [1].Detailed.element_data[15].prec_code := 3, [1].Detailed.element_data[15].Unit_code := 12, [1].Detailed.element_data[15].result_measurement := 5.231574, [2].UID := 43002, [2].Basic.unique_id := 43002, [2].Basic.channel_num := 1, [2].Basic.program_num := 2, [2].Basic.evaluation_code := 1, [2].Basic.test_port := 1, [2].Basic.year := 26, [2].Basic.month := 6, [2].Basic.date := 5, [2].Basic.hour := 10, [2].Basic.minute := 14, [2].Basic.second := 6, [2].Basic.flags := 12, [2].Basic.Num_tests := 1, [2].Basic.test_elements.test_type := 66,
        [2].Basic.test_elements.test_eval := 1, [2].Basic.test_elements.num_elements := 16, [2].Detailed.unique_id := 43002, [2].Detailed.num_elements := 16, [2].Detailed.Test_Type := 66, [2].Detailed.element_data[0].Variable_code := 61, [2].Detailed.element_data[0].prec_code := 2, [2].Detailed.element_data[0].Unit_code := 60, [2].Detailed.element_data[0].result_measurement := 0.007264316, [2].Detailed.element_data[1].Variable_code := 28, [2].Detailed.element_data[1].prec_code := 3, [2].Detailed.element_data[1].Unit_code := 41, [2].Detailed.element_data[1].result_measurement := 0.00016298145, [2].Detailed.element_data[2].Variable_code := 13, [2].Detailed.element_data[2].prec_code := 3, [2].Detailed.element_data[2].Unit_code := 12, [2].Detailed.element_data[2].result_measurement := 5.1514387, [2].Detailed.element_data[3].Variable_code := 75, [2].Detailed.element_data[3].prec_code := 2, [2].Detailed.element_data[3].Unit_code := 60, [2].Detailed.element_data[4].Variable_code := 60, [2].Detailed.element_data[4].prec_code := 2, [2].Detailed.element_data[4].Unit_code := 60, [2].Detailed.element_data[4].result_measurement := 0.0033527613, [2].Detailed.element_data[5].Variable_code := 56, [2].Detailed.element_data[5].prec_code := 3, [2].Detailed.element_data[5].Unit_code := 41, [2].Detailed.element_data[6].Variable_code := 55, [2].Detailed.element_data[6].prec_code := 3, [2].Detailed.element_data[6].Unit_code := 12, [2].Detailed.element_data[6].result_measurement := 5.1514387, [2].Detailed.element_data[7].Variable_code := 58, [2].Detailed.element_data[7].prec_code := 2, [2].Detailed.element_data[7].Unit_code := 60, [2].Detailed.element_data[7].result_measurement := -1.0002404, [2].Detailed.element_data[8].Variable_code := 59, [2].Detailed.element_data[8].prec_code := 2, [2].Detailed.element_data[8].Unit_code := 60, [2].Detailed.element_data[8].result_measurement := 1.0002404, [2].Detailed.element_data[9].Variable_code := 12, [2].Detailed.element_data[9].prec_code := 3, [2].Detailed.element_data[9].Unit_code := 12, [2].Detailed.element_data[9].result_measurement := 5.000001, [2].Detailed.element_data[10].Variable_code := 62, [2].Detailed.element_data[10].prec_code := 2, [2].Detailed.element_data[10].Unit_code := 60, [2].Detailed.element_data[10].result_measurement := 1.1298805, [2].Detailed.element_data[11].Variable_code := 21, [2].Detailed.element_data[11].prec_code := 3, [2].Detailed.element_data[11].Unit_code := 41, [2].Detailed.element_data[11].result_measurement := 4.656613e-06, [2].Detailed.element_data[12].Variable_code := 25, [2].Detailed.element_data[12].prec_code := 3, [2].Detailed.element_data[12].Unit_code := 41, [2].Detailed.element_data[12].result_measurement := 0.023245811, [2].Detailed.element_data[13].Variable_code := 216, [2].Detailed.element_data[13].prec_code := 3, [2].Detailed.element_data[13].Unit_code := 41, [2].Detailed.element_data[13].result_measurement := -3.7252903e-05, [2].Detailed.element_data[14].Variable_code := 218,
        [2].Detailed.element_data[14].prec_code := 3, [2].Detailed.element_data[14].Unit_code := 41, [2].Detailed.element_data[14].result_measurement := 0.011632219, [2].Detailed.element_data[15].Variable_code := 295, [2].Detailed.element_data[15].prec_code := 3, [2].Detailed.element_data[15].Unit_code := 12, [2].Detailed.element_data[15].result_measurement := 5.152752, [3].UID := 43008, [3].Basic.unique_id := 43008, [3].Basic.channel_num := 1, [3].Basic.program_num := 2, [3].Basic.evaluation_code := 1, [3].Basic.test_port := 1, [3].Basic.year := 26, [3].Basic.month := 6, [3].Basic.date := 5, [3].Basic.hour := 10, [3].Basic.minute := 17, [3].Basic.second := 58, [3].Basic.flags := 12, [3].Basic.Num_tests := 1, [3].Basic.test_elements.test_type := 66, [3].Basic.test_elements.test_eval := 1, [3].Basic.test_elements.num_elements := 16, [3].Detailed.unique_id := 43008, [3].Detailed.num_elements := 16, [3].Detailed.Test_Type := 66, [3].Detailed.element_data[0].Variable_code := 61, [3].Detailed.element_data[0].prec_code := 2, [3].Detailed.element_data[0].Unit_code := 60, [3].Detailed.element_data[0].result_measurement := 0.0067055225, [3].Detailed.element_data[1].Variable_code := 28, [3].Detailed.element_data[1].prec_code := 3, [3].Detailed.element_data[1].Unit_code := 41, [3].Detailed.element_data[1].result_measurement := 0.00014901161, [3].Detailed.element_data[2].Variable_code := 13, [3].Detailed.element_data[2].prec_code := 3, [3].Detailed.element_data[2].Unit_code := 12, [3].Detailed.element_data[2].result_measurement := 5.146321, [3].Detailed.element_data[3].Variable_code := 75, [3].Detailed.element_data[3].prec_code := 2, [3].Detailed.element_data[3].Unit_code := 60, [3].Detailed.element_data[4].Variable_code := 60, [3].Detailed.element_data[4].prec_code := 2, [3].Detailed.element_data[4].Unit_code := 60, [3].Detailed.element_data[4].result_measurement := 0.011734664, [3].Detailed.element_data[5].Variable_code := 56, [3].Detailed.element_data[5].prec_code := 3, [3].Detailed.element_data[5].Unit_code := 41, [3].Detailed.element_data[5].result_measurement := 8.8475645e-05, [3].Detailed.element_data[6].Variable_code := 55, [3].Detailed.element_data[6].prec_code := 3, [3].Detailed.element_data[6].Unit_code := 12, [3].Detailed.element_data[6].result_measurement := 5.146321, [3].Detailed.element_data[7].Variable_code := 58, [3].Detailed.element_data[7].prec_code := 2, [3].Detailed.element_data[7].Unit_code := 60, [3].Detailed.element_data[7].result_measurement := -1.0002404, [3].Detailed.element_data[8].Variable_code := 59, [3].Detailed.element_data[8].prec_code := 2,
        [3].Detailed.element_data[8].Unit_code := 60, [3].Detailed.element_data[8].result_measurement := 1.0002404, [3].Detailed.element_data[9].Variable_code := 12, [3].Detailed.element_data[9].prec_code := 3, [3].Detailed.element_data[9].Unit_code := 12, [3].Detailed.element_data[9].result_measurement := 5.000001, [3].Detailed.element_data[10].Variable_code := 62, [3].Detailed.element_data[10].prec_code := 2, [3].Detailed.element_data[10].Unit_code := 60, [3].Detailed.element_data[10].result_measurement := 1.1298805, [3].Detailed.element_data[11].Variable_code := 21, [3].Detailed.element_data[11].prec_code := 3, [3].Detailed.element_data[11].Unit_code := 41, [3].Detailed.element_data[11].result_measurement := 4.656613e-06, [3].Detailed.element_data[12].Variable_code := 25, [3].Detailed.element_data[12].prec_code := 3, [3].Detailed.element_data[12].Unit_code := 41, [3].Detailed.element_data[12].result_measurement := 0.023245811, [3].Detailed.element_data[13].Variable_code := 216, [3].Detailed.element_data[13].prec_code := 3, [3].Detailed.element_data[13].Unit_code := 41, [3].Detailed.element_data[13].result_measurement := -3.7252903e-05, [3].Detailed.element_data[14].Variable_code := 218, [3].Detailed.element_data[14].prec_code := 3, [3].Detailed.element_data[14].Unit_code := 41, [3].Detailed.element_data[14].result_measurement := 0.011632219, [3].Detailed.element_data[15].Variable_code := 295, [3].Detailed.element_data[15].prec_code := 3, [3].Detailed.element_data[15].Unit_code := 12, [3].Detailed.element_data[15].result_measurement := 5.1471496, [4].UID := 43011, [4].Basic.unique_id := 43011, [4].Basic.channel_num := 1, [4].Basic.program_num := 2, [4].Basic.evaluation_code := 1, [4].Basic.test_port := 1, [4].Basic.year := 26, [4].Basic.month := 6, [4].Basic.date := 5, [4].Basic.hour := 10, [4].Basic.minute := 18, [4].Basic.second := 57, [4].Basic.flags := 12, [4].Basic.Num_tests := 1, [4].Basic.test_elements.test_type := 66, [4].Basic.test_elements.test_eval := 1, [4].Basic.test_elements.num_elements := 16, [4].Detailed.unique_id := 43011, [4].Detailed.num_elements := 16, [4].Detailed.Test_Type := 66, [4].Detailed.element_data[0].Variable_code := 61, [4].Detailed.element_data[0].prec_code := 2, [4].Detailed.element_data[0].Unit_code := 60, [4].Detailed.element_data[0].result_measurement := -0.0033527613, [4].Detailed.element_data[1].Variable_code := 28, [4].Detailed.element_data[1].prec_code := 3, [4].Detailed.element_data[1].Unit_code := 41, [4].Detailed.element_data[1].result_measurement := -7.4505806e-05, [4].Detailed.element_data[2].Variable_code := 13, [4].Detailed.element_data[2].prec_code := 3,
        [4].Detailed.element_data[2].Unit_code := 12, [4].Detailed.element_data[2].result_measurement := 5.146088, [4].Detailed.element_data[3].Variable_code := 75, [4].Detailed.element_data[3].prec_code := 2, [4].Detailed.element_data[3].Unit_code := 60, [4].Detailed.element_data[4].Variable_code := 60, [4].Detailed.element_data[4].prec_code := 2, [4].Detailed.element_data[4].Unit_code := 60, [4].Detailed.element_data[4].result_measurement := 0.007264316, [4].Detailed.element_data[5].Variable_code := 56, [4].Detailed.element_data[5].prec_code := 3, [4].Detailed.element_data[5].Unit_code := 41, [4].Detailed.element_data[5].result_measurement := 4.1909516e-05, [4].Detailed.element_data[6].Variable_code := 55, [4].Detailed.element_data[6].prec_code := 3, [4].Detailed.element_data[6].Unit_code := 12, [4].Detailed.element_data[6].result_measurement := 5.146088, [4].Detailed.element_data[7].Variable_code := 58, [4].Detailed.element_data[7].prec_code := 2, [4].Detailed.element_data[7].Unit_code := 60, [4].Detailed.element_data[7].result_measurement := -1.0002404, [4].Detailed.element_data[8].Variable_code := 59, [4].Detailed.element_data[8].prec_code := 2, [4].Detailed.element_data[8].Unit_code := 60, [4].Detailed.element_data[8].result_measurement := 1.0002404, [4].Detailed.element_data[9].Variable_code := 12, [4].Detailed.element_data[9].prec_code := 3, [4].Detailed.element_data[9].Unit_code := 12, [4].Detailed.element_data[9].result_measurement := 5.000001, [4].Detailed.element_data[10].Variable_code := 62, [4].Detailed.element_data[10].prec_code := 2, [4].Detailed.element_data[10].Unit_code := 60, [4].Detailed.element_data[10].result_measurement := 1.1298805, [4].Detailed.element_data[11].Variable_code := 21, [4].Detailed.element_data[11].prec_code := 3, [4].Detailed.element_data[11].Unit_code := 41, [4].Detailed.element_data[11].result_measurement := 4.656613e-06, [4].Detailed.element_data[12].Variable_code := 25, [4].Detailed.element_data[12].prec_code := 3, [4].Detailed.element_data[12].Unit_code := 41, [4].Detailed.element_data[12].result_measurement := 0.023245811, [4].Detailed.element_data[13].Variable_code := 216, [4].Detailed.element_data[13].prec_code := 3, [4].Detailed.element_data[13].Unit_code := 41, [4].Detailed.element_data[13].result_measurement := -3.7252903e-05, [4].Detailed.element_data[14].Variable_code := 218, [4].Detailed.element_data[14].prec_code := 3, [4].Detailed.element_data[14].Unit_code := 41, [4].Detailed.element_data[14].result_measurement := 0.011632219, [4].Detailed.element_data[15].Variable_code := 295, [4].Detailed.element_data[15].prec_code := 3, [4].Detailed.element_data[15].Unit_code := 12, [4].Detailed.element_data[15].result_measurement := 5.147038, [5].UID := 43014, [5].Basic.unique_id := 43014, [5].Basic.channel_num := 1, [5].Basic.program_num := 2, [5].Basic.evaluation_code := 1, [5].Basic.test_port := 1, [5].Basic.year := 26,
        [5].Basic.month := 6, [5].Basic.date := 5, [5].Basic.hour := 10, [5].Basic.minute := 19, [5].Basic.second := 51, [5].Basic.flags := 12, [5].Basic.Num_tests := 1, [5].Basic.test_elements.test_type := 66, [5].Basic.test_elements.test_eval := 1, [5].Basic.test_elements.num_elements := 16, [5].Detailed.unique_id := 43014, [5].Detailed.num_elements := 16, [5].Detailed.Test_Type := 66, [5].Detailed.element_data[0].Variable_code := 61, [5].Detailed.element_data[0].prec_code := 2, [5].Detailed.element_data[0].Unit_code := 60, [5].Detailed.element_data[0].result_measurement := 0.007264316, [5].Detailed.element_data[1].Variable_code := 28, [5].Detailed.element_data[1].prec_code := 3, [5].Detailed.element_data[1].Unit_code := 41, [5].Detailed.element_data[1].result_measurement := 0.00015832484, [5].Detailed.element_data[2].Variable_code := 13, [5].Detailed.element_data[2].prec_code := 3, [5].Detailed.element_data[2].Unit_code := 12, [5].Detailed.element_data[2].result_measurement := 5.146228, [5].Detailed.element_data[3].Variable_code := 75, [5].Detailed.element_data[3].prec_code := 2, [5].Detailed.element_data[3].Unit_code := 60, [5].Detailed.element_data[4].Variable_code := 60, [5].Detailed.element_data[4].prec_code := 2, [5].Detailed.element_data[4].Unit_code := 60, [5].Detailed.element_data[4].result_measurement := 0.014528632, [5].Detailed.element_data[5].Variable_code := 56, [5].Detailed.element_data[5].prec_code := 3, [5].Detailed.element_data[5].Unit_code := 41, [5].Detailed.element_data[5].result_measurement := 0.00011641532, [5].Detailed.element_data[6].Variable_code := 55, [5].Detailed.element_data[6].prec_code := 3, [5].Detailed.element_data[6].Unit_code := 12, [5].Detailed.element_data[6].result_measurement := 5.146228, [5].Detailed.element_data[7].Variable_code := 58, [5].Detailed.element_data[7].prec_code := 2, [5].Detailed.element_data[7].Unit_code := 60, [5].Detailed.element_data[7].result_measurement := -1.0002404, [5].Detailed.element_data[8].Variable_code := 59, [5].Detailed.element_data[8].prec_code := 2, [5].Detailed.element_data[8].Unit_code := 60, [5].Detailed.element_data[8].result_measurement := 1.0002404, [5].Detailed.element_data[9].Variable_code := 12, [5].Detailed.element_data[9].prec_code := 3, [5].Detailed.element_data[9].Unit_code := 12, [5].Detailed.element_data[9].result_measurement := 5.000001, [5].Detailed.element_data[10].Variable_code := 62, [5].Detailed.element_data[10].prec_code := 2, [5].Detailed.element_data[10].Unit_code := 60, [5].Detailed.element_data[10].result_measurement := 1.1298805, [5].Detailed.element_data[11].Variable_code := 21, [5].Detailed.element_data[11].prec_code := 3, [5].Detailed.element_data[11].Unit_code := 41, [5].Detailed.element_data[11].result_measurement := 4.656613e-06,
        [5].Detailed.element_data[12].Variable_code := 25, [5].Detailed.element_data[12].prec_code := 3, [5].Detailed.element_data[12].Unit_code := 41, [5].Detailed.element_data[12].result_measurement := 0.023245811, [5].Detailed.element_data[13].Variable_code := 216, [5].Detailed.element_data[13].prec_code := 3, [5].Detailed.element_data[13].Unit_code := 41, [5].Detailed.element_data[13].result_measurement := -3.7252903e-05, [5].Detailed.element_data[14].Variable_code := 218, [5].Detailed.element_data[14].prec_code := 3, [5].Detailed.element_data[14].Unit_code := 41, [5].Detailed.element_data[14].result_measurement := 0.011632219, [5].Detailed.element_data[15].Variable_code := 295, [5].Detailed.element_data[15].prec_code := 3, [5].Detailed.element_data[15].Unit_code := 12, [5].Detailed.element_data[15].result_measurement := 5.14742, [7].UID := 9472, [7].Basic.unique_id := 9472, [7].Basic.channel_num := 1, [7].Basic.program_num := 2, [7].Basic.evaluation_code := 1, [7].Basic.test_port := 1, [7].Basic.year := 26, [7].Basic.month := 9, [7].Basic.date := 24, [7].Basic.hour := 19, [7].Basic.minute := 43, [7].Basic.second := 44, [7].Basic.flags := 12, [7].Basic.Num_tests := 1, [7].Basic.test_elements.test_type := 66, [7].Basic.test_elements.test_eval := 1, [7].Basic.test_elements.num_elements := 16, [7].Detailed.unique_id := 9472, [7].Detailed.num_elements := 16, [7].Detailed.Test_Type := 66, [7].Detailed.element_data[0].Variable_code := 61, [7].Detailed.element_data[0].prec_code := 2, [7].Detailed.element_data[0].Unit_code := 60, [7].Detailed.element_data[0].result_measurement := -0.045262277, [7].Detailed.element_data[1].Variable_code := 28, [7].Detailed.element_data[1].prec_code := 3, [7].Detailed.element_data[1].Unit_code := 41, [7].Detailed.element_data[1].result_measurement := 0.00067520887, [7].Detailed.element_data[2].Variable_code := 13, [7].Detailed.element_data[2].prec_code := 3, [7].Detailed.element_data[2].Unit_code := 12, [7].Detailed.element_data[2].result_measurement := 5.060546, [7].Detailed.element_data[3].Variable_code := 75, [7].Detailed.element_data[3].prec_code := 2, [7].Detailed.element_data[3].Unit_code := 60, [7].Detailed.element_data[4].Variable_code := 60, [7].Detailed.element_data[4].prec_code := 2, [7].Detailed.element_data[4].Unit_code := 60, [7].Detailed.element_data[4].result_measurement := -0.07208437, [7].Detailed.element_data[5].Variable_code := 56, [7].Detailed.element_data[5].prec_code := 3, [7].Detailed.element_data[5].Unit_code := 41, [7].Detailed.element_data[5].result_measurement := 0.00018626451, [7].Detailed.element_data[6].Variable_code := 55,
        [7].Detailed.element_data[6].prec_code := 3, [7].Detailed.element_data[6].Unit_code := 12, [7].Detailed.element_data[6].result_measurement := 5.060546, [7].Detailed.element_data[7].Variable_code := 58, [7].Detailed.element_data[7].prec_code := 2, [7].Detailed.element_data[7].Unit_code := 60, [7].Detailed.element_data[7].result_measurement := -1.0002404, [7].Detailed.element_data[8].Variable_code := 59, [7].Detailed.element_data[8].prec_code := 2, [7].Detailed.element_data[8].Unit_code := 60, [7].Detailed.element_data[8].result_measurement := 1.0002404, [7].Detailed.element_data[9].Variable_code := 12, [7].Detailed.element_data[9].prec_code := 3, [7].Detailed.element_data[9].Unit_code := 12, [7].Detailed.element_data[9].result_measurement := 5.000001, [7].Detailed.element_data[10].Variable_code := 62, [7].Detailed.element_data[10].prec_code := 2, [7].Detailed.element_data[10].Unit_code := 60, [7].Detailed.element_data[10].result_measurement := 1.0902061, [7].Detailed.element_data[11].Variable_code := 21, [7].Detailed.element_data[11].prec_code := 3, [7].Detailed.element_data[11].Unit_code := 41, [7].Detailed.element_data[11].result_measurement := 0.0015180558, [7].Detailed.element_data[12].Variable_code := 25, [7].Detailed.element_data[12].prec_code := 3, [7].Detailed.element_data[12].Unit_code := 41, [7].Detailed.element_data[12].result_measurement := 0.021727756, [7].Detailed.element_data[13].Variable_code := 216, [7].Detailed.element_data[13].prec_code := 3, [7].Detailed.element_data[13].Unit_code := 41, [7].Detailed.element_data[13].result_measurement := 0.00085681677, [7].Detailed.element_data[14].Variable_code := 218, [7].Detailed.element_data[14].prec_code := 3, [7].Detailed.element_data[14].Unit_code := 41, [7].Detailed.element_data[14].result_measurement := 0.01094304, [7].Detailed.element_data[15].Variable_code := 295, [7].Detailed.element_data[15].prec_code := 3, [7].Detailed.element_data[15].Unit_code := 12, [7].Detailed.element_data[15].result_measurement := 5.0637546, [8].UID := 9475, [8].Basic.unique_id := 9475, [8].Basic.channel_num := 1, [8].Basic.program_num := 2, [8].Basic.evaluation_code := 1, [8].Basic.test_port := 1, [8].Basic.year := 26, [8].Basic.month := 9, [8].Basic.date := 24, [8].Basic.hour := 19, [8].Basic.minute := 46, [8].Basic.second := 23, [8].Basic.flags := 12, [8].Basic.Num_tests := 1, [8].Basic.test_elements.test_type := 66, [8].Basic.test_elements.test_eval := 1, [8].Basic.test_elements.num_elements := 16, [8].Detailed.unique_id := 9475, [8].Detailed.num_elements := 16, [8].Detailed.Test_Type := 66, [8].Detailed.element_data[0].Variable_code := 61,
        [8].Detailed.element_data[0].prec_code := 2, [8].Detailed.element_data[0].Unit_code := 60, [8].Detailed.element_data[0].result_measurement := -0.029616058, [8].Detailed.element_data[1].Variable_code := 28, [8].Detailed.element_data[1].prec_code := 3, [8].Detailed.element_data[1].Unit_code := 41, [8].Detailed.element_data[1].result_measurement := 0.0009685755, [8].Detailed.element_data[2].Variable_code := 13, [8].Detailed.element_data[2].prec_code := 3, [8].Detailed.element_data[2].Unit_code := 12, [8].Detailed.element_data[2].result_measurement := 5.059587, [8].Detailed.element_data[3].Variable_code := 75, [8].Detailed.element_data[3].prec_code := 2, [8].Detailed.element_data[3].Unit_code := 60, [8].Detailed.element_data[4].Variable_code := 60, [8].Detailed.element_data[4].prec_code := 2, [8].Detailed.element_data[4].Unit_code := 60, [8].Detailed.element_data[4].result_measurement := -0.03799796, [8].Detailed.element_data[5].Variable_code := 56, [8].Detailed.element_data[5].prec_code := 3, [8].Detailed.element_data[5].Unit_code := 41, [8].Detailed.element_data[5].result_measurement := 0.0005029142, [8].Detailed.element_data[6].Variable_code := 55, [8].Detailed.element_data[6].prec_code := 3, [8].Detailed.element_data[6].Unit_code := 12, [8].Detailed.element_data[6].result_measurement := 5.059587, [8].Detailed.element_data[7].Variable_code := 58, [8].Detailed.element_data[7].prec_code := 2, [8].Detailed.element_data[7].Unit_code := 60, [8].Detailed.element_data[7].result_measurement := -1.0002404, [8].Detailed.element_data[8].Variable_code := 59, [8].Detailed.element_data[8].prec_code := 2, [8].Detailed.element_data[8].Unit_code := 60, [8].Detailed.element_data[8].result_measurement := 1.0002404, [8].Detailed.element_data[9].Variable_code := 12, [8].Detailed.element_data[9].prec_code := 3, [8].Detailed.element_data[9].Unit_code := 12, [8].Detailed.element_data[9].result_measurement := 5.000001, [8].Detailed.element_data[10].Variable_code := 62, [8].Detailed.element_data[10].prec_code := 2, [8].Detailed.element_data[10].Unit_code := 60, [8].Detailed.element_data[10].result_measurement := 1.0902061, [8].Detailed.element_data[11].Variable_code := 21, [8].Detailed.element_data[11].prec_code := 3, [8].Detailed.element_data[11].Unit_code := 41, [8].Detailed.element_data[11].result_measurement := 0.0015180558, [8].Detailed.element_data[12].Variable_code := 25, [8].Detailed.element_data[12].prec_code := 3, [8].Detailed.element_data[12].Unit_code := 41, [8].Detailed.element_data[12].result_measurement := 0.021727756, [8].Detailed.element_data[13].Variable_code := 216, [8].Detailed.element_data[13].prec_code := 3, [8].Detailed.element_data[13].Unit_code := 41, [8].Detailed.element_data[13].result_measurement := 0.00085681677, [8].Detailed.element_data[14].Variable_code := 218, [8].Detailed.element_data[14].prec_code := 3, [8].Detailed.element_data[14].Unit_code := 41, [8].Detailed.element_data[14].result_measurement := 0.01094304, [8].Detailed.element_data[15].Variable_code := 295, [8].Detailed.element_data[15].prec_code := 3,
        [8].Detailed.element_data[15].Unit_code := 12, [8].Detailed.element_data[15].result_measurement := 5.062413, [9].UID := 9478, [9].Basic.unique_id := 9478, [9].Basic.channel_num := 1, [9].Basic.program_num := 2, [9].Basic.evaluation_code := 1, [9].Basic.test_port := 1, [9].Basic.year := 26, [9].Basic.month := 9, [9].Basic.date := 24, [9].Basic.hour := 19, [9].Basic.minute := 52, [9].Basic.second := 10, [9].Basic.flags := 12, [9].Basic.Num_tests := 1, [9].Basic.test_elements.test_type := 66, [9].Basic.test_elements.test_eval := 1, [9].Basic.test_elements.num_elements := 16, [9].Detailed.unique_id := 9478, [9].Detailed.num_elements := 16, [9].Detailed.Test_Type := 66, [9].Detailed.element_data[0].Variable_code := 61, [9].Detailed.element_data[0].prec_code := 2, [9].Detailed.element_data[0].Unit_code := 60, [9].Detailed.element_data[0].result_measurement := -0.051409006, [9].Detailed.element_data[1].Variable_code := 28, [9].Detailed.element_data[1].prec_code := 3, [9].Detailed.element_data[1].Unit_code := 41, [9].Detailed.element_data[1].result_measurement := 0.00056345016, [9].Detailed.element_data[2].Variable_code := 13, [9].Detailed.element_data[2].prec_code := 3, [9].Detailed.element_data[2].Unit_code := 12, [9].Detailed.element_data[2].result_measurement := 5.0597124, [9].Detailed.element_data[3].Variable_code := 75, [9].Detailed.element_data[3].prec_code := 2, [9].Detailed.element_data[3].Unit_code := 60, [9].Detailed.element_data[4].Variable_code := 60, [9].Detailed.element_data[4].prec_code := 2, [9].Detailed.element_data[4].Unit_code := 60, [9].Detailed.element_data[4].result_measurement := -0.08158386, [9].Detailed.element_data[5].Variable_code := 56, [9].Detailed.element_data[5].prec_code := 3, [9].Detailed.element_data[5].Unit_code := 41, [9].Detailed.element_data[5].result_measurement := 9.778887e-05, [9].Detailed.element_data[6].Variable_code := 55, [9].Detailed.element_data[6].prec_code := 3, [9].Detailed.element_data[6].Unit_code := 12, [9].Detailed.element_data[6].result_measurement := 5.0597124, [9].Detailed.element_data[7].Variable_code := 58, [9].Detailed.element_data[7].prec_code := 2, [9].Detailed.element_data[7].Unit_code := 60, [9].Detailed.element_data[7].result_measurement := -1.0002404, [9].Detailed.element_data[8].Variable_code := 59, [9].Detailed.element_data[8].prec_code := 2, [9].Detailed.element_data[8].Unit_code := 60, [9].Detailed.element_data[8].result_measurement := 1.0002404, [9].Detailed.element_data[9].Variable_code := 12, [9].Detailed.element_data[9].prec_code := 3, [9].Detailed.element_data[9].Unit_code := 12,
        [9].Detailed.element_data[9].result_measurement := 5.000001, [9].Detailed.element_data[10].Variable_code := 62, [9].Detailed.element_data[10].prec_code := 2, [9].Detailed.element_data[10].Unit_code := 60, [9].Detailed.element_data[10].result_measurement := 1.0902061, [9].Detailed.element_data[11].Variable_code := 21, [9].Detailed.element_data[11].prec_code := 3, [9].Detailed.element_data[11].Unit_code := 41, [9].Detailed.element_data[11].result_measurement := 0.0015180558, [9].Detailed.element_data[12].Variable_code := 25, [9].Detailed.element_data[12].prec_code := 3, [9].Detailed.element_data[12].Unit_code := 41, [9].Detailed.element_data[12].result_measurement := 0.021727756, [9].Detailed.element_data[13].Variable_code := 216, [9].Detailed.element_data[13].prec_code := 3, [9].Detailed.element_data[13].Unit_code := 41, [9].Detailed.element_data[13].result_measurement := 0.00085681677, [9].Detailed.element_data[14].Variable_code := 218, [9].Detailed.element_data[14].prec_code := 3, [9].Detailed.element_data[14].Unit_code := 41, [9].Detailed.element_data[14].result_measurement := 0.01094304, [9].Detailed.element_data[15].Variable_code := 295, [9].Detailed.element_data[15].prec_code := 3, [9].Detailed.element_data[15].Unit_code := 12, [9].Detailed.element_data[15].result_measurement := 5.063093);
   CTS1_ResultHistoryVol : udt_CTS_RESULT[10] := ([0].UID := 43004, [0].Basic.unique_id := 43004, [0].Basic.channel_num := 1, [0].Basic.program_num := 1, [0].Basic.evaluation_code := 1, [0].Basic.test_port := 1, [0].Basic.year := 26, [0].Basic.month := 6, [0].Basic.date := 5, [0].Basic.hour := 10, [0].Basic.minute := 17, [0].Basic.second := 10, [0].Basic.flags := 12, [0].Basic.Num_tests := 1, [0].Basic.test_elements.test_type := 69, [0].Basic.test_elements.test_eval := 1, [0].Basic.test_elements.num_elements := 4, [0].Detailed.unique_id := 43004, [0].Detailed.num_elements := 4, [0].Detailed.Test_Type := 69, [0].Detailed.element_data[0].Variable_code := 245, [0].Detailed.element_data[0].prec_code := 2, [0].Detailed.element_data[0].Unit_code := 165, [0].Detailed.element_data[0].result_measurement := 187.00204, [0].Detailed.element_data[1].Variable_code := 13, [0].Detailed.element_data[1].prec_code := 3, [0].Detailed.element_data[1].Unit_code := 12, [0].Detailed.element_data[1].result_measurement := 1.779967, [0].Detailed.element_data[2].Variable_code := 247, [0].Detailed.element_data[2].prec_code := 3, [0].Detailed.element_data[2].Unit_code := 12, [0].Detailed.element_data[2].result_measurement := 5.108542, [0].Detailed.element_data[3].Variable_code := 295, [0].Detailed.element_data[3].prec_code := 3, [0].Detailed.element_data[3].Unit_code := 12, [0].Detailed.element_data[3].result_measurement := 5.1097245, [1].UID := 43007, [1].Basic.unique_id := 43007, [1].Basic.channel_num := 1, [1].Basic.program_num := 1, [1].Basic.evaluation_code := 1, [1].Basic.test_port := 1, [1].Basic.year := 26, [1].Basic.month := 6, [1].Basic.date := 5, [1].Basic.hour := 10, [1].Basic.minute := 17, [1].Basic.second := 51, [1].Basic.flags := 12, [1].Basic.Num_tests := 1, [1].Basic.test_elements.test_type := 69, [1].Basic.test_elements.test_eval := 1, [1].Basic.test_elements.num_elements := 4, [1].Detailed.unique_id := 43007, [1].Detailed.num_elements := 4, [1].Detailed.Test_Type := 69, [1].Detailed.element_data[0].Variable_code := 245, [1].Detailed.element_data[0].prec_code := 2, [1].Detailed.element_data[0].Unit_code := 165, [1].Detailed.element_data[0].result_measurement := 187.18288,
        [1].Detailed.element_data[1].Variable_code := 13, [1].Detailed.element_data[1].prec_code := 3, [1].Detailed.element_data[1].Unit_code := 12, [1].Detailed.element_data[1].result_measurement := 1.7796829, [1].Detailed.element_data[2].Variable_code := 247, [1].Detailed.element_data[2].prec_code := 3, [1].Detailed.element_data[2].Unit_code := 12, [1].Detailed.element_data[2].result_measurement := 5.1109447, [1].Detailed.element_data[3].Variable_code := 295, [1].Detailed.element_data[3].prec_code := 3, [1].Detailed.element_data[3].Unit_code := 12, [1].Detailed.element_data[3].result_measurement := 5.112132, [2].UID := 43010, [2].Basic.unique_id := 43010, [2].Basic.channel_num := 1, [2].Basic.program_num := 1, [2].Basic.evaluation_code := 1, [2].Basic.test_port := 1, [2].Basic.year := 26, [2].Basic.month := 6, [2].Basic.date := 5, [2].Basic.hour := 10, [2].Basic.minute := 18, [2].Basic.second := 50, [2].Basic.flags := 12, [2].Basic.Num_tests := 1, [2].Basic.test_elements.test_type := 69, [2].Basic.test_elements.test_eval := 1, [2].Basic.test_elements.num_elements := 4, [2].Detailed.unique_id := 43010, [2].Detailed.num_elements := 4, [2].Detailed.Test_Type := 69, [2].Detailed.element_data[0].Variable_code := 245, [2].Detailed.element_data[0].prec_code := 2, [2].Detailed.element_data[0].Unit_code := 165, [2].Detailed.element_data[0].result_measurement := 187.18771, [2].Detailed.element_data[1].Variable_code := 13, [2].Detailed.element_data[1].prec_code := 3, [2].Detailed.element_data[1].Unit_code := 12, [2].Detailed.element_data[1].result_measurement := 1.7792639, [2].Detailed.element_data[2].Variable_code := 247, [2].Detailed.element_data[2].prec_code := 3, [2].Detailed.element_data[2].Unit_code := 12, [2].Detailed.element_data[2].result_measurement := 5.109827, [2].Detailed.element_data[3].Variable_code := 295, [2].Detailed.element_data[3].prec_code := 3, [2].Detailed.element_data[3].Unit_code := 12, [2].Detailed.element_data[3].result_measurement := 5.1112704, [3].UID := 43013, [3].Basic.unique_id := 43013, [3].Basic.channel_num := 1, [3].Basic.program_num := 1, [3].Basic.evaluation_code := 1, [3].Basic.test_port := 1, [3].Basic.year := 26, [3].Basic.month := 6, [3].Basic.date := 5, [3].Basic.hour := 10, [3].Basic.minute := 19, [3].Basic.second := 44,
        [3].Basic.flags := 12, [3].Basic.Num_tests := 1, [3].Basic.test_elements.test_type := 69, [3].Basic.test_elements.test_eval := 1, [3].Basic.test_elements.num_elements := 4, [3].Detailed.unique_id := 43013, [3].Detailed.num_elements := 4, [3].Detailed.Test_Type := 69, [3].Detailed.element_data[0].Variable_code := 245, [3].Detailed.element_data[0].prec_code := 2, [3].Detailed.element_data[0].Unit_code := 165, [3].Detailed.element_data[0].result_measurement := 187.24707, [3].Detailed.element_data[1].Variable_code := 13, [3].Detailed.element_data[1].prec_code := 3, [3].Detailed.element_data[1].Unit_code := 12, [3].Detailed.element_data[1].result_measurement := 1.7789285, [3].Detailed.element_data[2].Variable_code := 247, [3].Detailed.element_data[2].prec_code := 3, [3].Detailed.element_data[2].Unit_code := 12, [3].Detailed.element_data[2].result_measurement := 5.10992, [3].Detailed.element_data[3].Variable_code := 295, [3].Detailed.element_data[3].prec_code := 3, [3].Detailed.element_data[3].Unit_code := 12, [3].Detailed.element_data[3].result_measurement := 5.111359, [4].UID := 43016, [4].Basic.unique_id := 43016, [4].Basic.channel_num := 1, [4].Basic.program_num := 1, [4].Basic.evaluation_code := 1, [4].Basic.test_port := 1, [4].Basic.year := 26, [4].Basic.month := 6, [4].Basic.date := 5, [4].Basic.hour := 10, [4].Basic.minute := 54, [4].Basic.second := 35, [4].Basic.flags := 12, [4].Basic.Num_tests := 1, [4].Basic.test_elements.test_type := 69, [4].Basic.test_elements.test_eval := 1, [4].Basic.test_elements.num_elements := 4, [4].Detailed.unique_id := 43016, [4].Detailed.num_elements := 4, [4].Detailed.Test_Type := 69, [4].Detailed.element_data[0].Variable_code := 245, [4].Detailed.element_data[0].prec_code := 2, [4].Detailed.element_data[0].Unit_code := 165, [4].Detailed.element_data[0].result_measurement := 187.26138, [4].Detailed.element_data[1].Variable_code := 13, [4].Detailed.element_data[1].prec_code := 3, [4].Detailed.element_data[1].Unit_code := 12, [4].Detailed.element_data[1].result_measurement := 1.7757015, [4].Detailed.element_data[2].Variable_code := 247, [4].Detailed.element_data[2].prec_code := 3, [4].Detailed.element_data[2].Unit_code := 12, [4].Detailed.element_data[2].result_measurement := 5.100905, [4].Detailed.element_data[3].Variable_code := 295, [4].Detailed.element_data[3].prec_code := 3, [4].Detailed.element_data[3].Unit_code := 12, [4].Detailed.element_data[3].result_measurement := 5.1019387,
        [5].UID := 43019, [5].Basic.unique_id := 43019, [5].Basic.channel_num := 1, [5].Basic.program_num := 1, [5].Basic.evaluation_code := 1, [5].Basic.test_port := 1, [5].Basic.year := 26, [5].Basic.month := 6, [5].Basic.date := 5, [5].Basic.hour := 10, [5].Basic.minute := 54, [5].Basic.second := 59, [5].Basic.flags := 12, [5].Basic.Num_tests := 1, [5].Basic.test_elements.test_type := 69, [5].Basic.test_elements.test_eval := 1, [5].Basic.test_elements.num_elements := 4, [5].Detailed.unique_id := 43019, [5].Detailed.num_elements := 4, [5].Detailed.Test_Type := 69, [5].Detailed.element_data[0].Variable_code := 245, [5].Detailed.element_data[0].prec_code := 2, [5].Detailed.element_data[0].Unit_code := 165, [5].Detailed.element_data[0].result_measurement := 187.70357, [5].Detailed.element_data[1].Variable_code := 13, [5].Detailed.element_data[1].prec_code := 3, [5].Detailed.element_data[1].Unit_code := 12, [5].Detailed.element_data[1].result_measurement := 1.7710496, [5].Detailed.element_data[2].Variable_code := 247, [5].Detailed.element_data[2].prec_code := 3, [5].Detailed.element_data[2].Unit_code := 12, [5].Detailed.element_data[2].result_measurement := 5.0953727, [5].Detailed.element_data[3].Variable_code := 295, [5].Detailed.element_data[3].prec_code := 3, [5].Detailed.element_data[3].Unit_code := 12, [5].Detailed.element_data[3].result_measurement := 5.096975, [6].UID := 43022, [6].Basic.unique_id := 43022, [6].Basic.channel_num := 1, [6].Basic.program_num := 1, [6].Basic.evaluation_code := 2, [6].Basic.test_port := 1, [6].Basic.year := 26, [6].Basic.month := 6, [6].Basic.date := 5, [6].Basic.hour := 10, [6].Basic.minute := 56, [6].Basic.second := 7, [6].Basic.flags := 12, [6].Basic.Num_tests := 1, [6].Basic.test_elements.test_type := 69, [6].Basic.test_elements.test_eval := 2, [6].Basic.test_elements.num_elements := 4, [6].Detailed.unique_id := 43022, [6].Detailed.num_elements := 4, [6].Detailed.Test_Type := 69, [6].Detailed.element_data[0].Variable_code := 245, [6].Detailed.element_data[0].prec_code := 2, [6].Detailed.element_data[0].Unit_code := 165, [6].Detailed.element_data[0].result_measurement := 1000.0,
        [6].Detailed.element_data[1].Variable_code := 13, [6].Detailed.element_data[1].prec_code := 3, [6].Detailed.element_data[1].Unit_code := 12, [6].Detailed.element_data[1].result_measurement := 0.0047218055, [6].Detailed.element_data[2].Variable_code := 247, [6].Detailed.element_data[2].prec_code := 3, [6].Detailed.element_data[2].Unit_code := 12, [6].Detailed.element_data[2].result_measurement := 5.095699, [6].Detailed.element_data[3].Variable_code := 295, [6].Detailed.element_data[3].prec_code := 3, [6].Detailed.element_data[3].Unit_code := 12, [6].Detailed.element_data[3].result_measurement := 5.096928, [7].UID := 9471, [7].Basic.unique_id := 9471, [7].Basic.channel_num := 1, [7].Basic.program_num := 1, [7].Basic.evaluation_code := 1, [7].Basic.test_port := 1, [7].Basic.year := 26, [7].Basic.month := 9, [7].Basic.date := 24, [7].Basic.hour := 19, [7].Basic.minute := 43, [7].Basic.second := 38, [7].Basic.flags := 12, [7].Basic.Num_tests := 1, [7].Basic.test_elements.test_type := 69, [7].Basic.test_elements.test_eval := 1, [7].Basic.test_elements.num_elements := 4, [7].Detailed.unique_id := 9471, [7].Detailed.num_elements := 4, [7].Detailed.Test_Type := 69, [7].Detailed.element_data[0].Variable_code := 245, [7].Detailed.element_data[0].prec_code := 2, [7].Detailed.element_data[0].Unit_code := 165, [7].Detailed.element_data[0].result_measurement := 159.4703, [7].Detailed.element_data[1].Variable_code := 13, [7].Detailed.element_data[1].prec_code := 3, [7].Detailed.element_data[1].Unit_code := 12, [7].Detailed.element_data[1].result_measurement := 1.9419706, [7].Detailed.element_data[2].Variable_code := 247, [7].Detailed.element_data[2].prec_code := 3, [7].Detailed.element_data[2].Unit_code := 12, [7].Detailed.element_data[2].result_measurement := 5.038837, [7].Detailed.element_data[3].Variable_code := 295, [7].Detailed.element_data[3].prec_code := 3, [7].Detailed.element_data[3].Unit_code := 12, [7].Detailed.element_data[3].result_measurement := 5.0408535, [8].UID := 9474, [8].Basic.unique_id := 9474, [8].Basic.channel_num := 1, [8].Basic.program_num := 1, [8].Basic.evaluation_code := 1, [8].Basic.test_port := 1, [8].Basic.year := 26, [8].Basic.month := 9, [8].Basic.date := 24, [8].Basic.hour := 19, [8].Basic.minute := 46, [8].Basic.second := 16,
        [8].Basic.flags := 12, [8].Basic.Num_tests := 1, [8].Basic.test_elements.test_type := 69, [8].Basic.test_elements.test_eval := 1, [8].Basic.test_elements.num_elements := 4, [8].Detailed.unique_id := 9474, [8].Detailed.num_elements := 4, [8].Detailed.Test_Type := 69, [8].Detailed.element_data[0].Variable_code := 245, [8].Detailed.element_data[0].prec_code := 2, [8].Detailed.element_data[0].Unit_code := 165, [8].Detailed.element_data[0].result_measurement := 159.83955, [8].Detailed.element_data[1].Variable_code := 13, [8].Detailed.element_data[1].prec_code := 3, [8].Detailed.element_data[1].Unit_code := 12, [8].Detailed.element_data[1].result_measurement := 1.9387808, [8].Detailed.element_data[2].Variable_code := 247, [8].Detailed.element_data[2].prec_code := 3, [8].Detailed.element_data[2].Unit_code := 12, [8].Detailed.element_data[2].result_measurement := 5.0377192, [8].Detailed.element_data[3].Variable_code := 295, [8].Detailed.element_data[3].prec_code := 3, [8].Detailed.element_data[3].Unit_code := 12, [8].Detailed.element_data[3].result_measurement := 5.0395913, [9].UID := 9477, [9].Basic.unique_id := 9477, [9].Basic.channel_num := 1, [9].Basic.program_num := 1, [9].Basic.evaluation_code := 1, [9].Basic.test_port := 1, [9].Basic.year := 26, [9].Basic.month := 9, [9].Basic.date := 24, [9].Basic.hour := 19, [9].Basic.minute := 52, [9].Basic.second := 3, [9].Basic.flags := 12, [9].Basic.Num_tests := 1, [9].Basic.test_elements.test_type := 69, [9].Basic.test_elements.test_eval := 1, [9].Basic.test_elements.num_elements := 4, [9].Detailed.unique_id := 9477, [9].Detailed.num_elements := 4, [9].Detailed.Test_Type := 69, [9].Detailed.element_data[0].Variable_code := 245, [9].Detailed.element_data[0].prec_code := 2, [9].Detailed.element_data[0].Unit_code := 165, [9].Detailed.element_data[0].result_measurement := 159.86131, [9].Detailed.element_data[1].Variable_code := 13, [9].Detailed.element_data[1].prec_code := 3, [9].Detailed.element_data[1].Unit_code := 12, [9].Detailed.element_data[1].result_measurement := 1.9387761, [9].Detailed.element_data[2].Variable_code := 247, [9].Detailed.element_data[2].prec_code := 3, [9].Detailed.element_data[2].Unit_code := 12, [9].Detailed.element_data[2].result_measurement := 5.0381293, [9].Detailed.element_data[3].Variable_code := 295, [9].Detailed.element_data[3].prec_code := 3, [9].Detailed.element_data[3].Unit_code := 12, [9].Detailed.element_data[3].result_measurement := 5.0394516);
   CTS1_Seq : udt_SequenceStructure_X64 := (CycleDone := 1, CurrentStep := 9000, NextStep := 9000, ONS := -32767, StepHistory[0] := 1030, StepHistory[1] := 2000, StepHistory[2] := 2010, StepHistory[3] := 2020, StepHistory[4] := 2030, StepHistory[5] := 9000, StepHistory[6] := 1000, StepHistory[7] := 1010, StepHistory[8] := 1020, StepHistory[9] := 9000, StepHistory[10] := 1000, StepHistory[11] := 1010, StepHistory[12] := 1020, StepHistory[13] := 9000, StepHistory[14] := 1000, StepHistory[15] := 1010, StepHistory[16] := 1020, StepHistory[17] := 9000, StepHistory[18] := 1000, StepHistory[19] := 1010, StepHistory[20] := 1020, StepHistory[21] := 9000, StepHistory[22] := 1000, StepHistory[23] := 1010, StepHistory[24] := 1020, StepHistory[25] := 9000, StepHistory[26] := 1000, StepHistory[27] := 1010, StepHistory[28] := 1020, StepHistory[29] := 1030, StepHistory[30] := 2000, StepHistory[31] := 2010, StepHistory[32] := 2020, StepHistory[33] := 2030, StepHistory[34] := 2000, StepHistory[35] := 2010, StepHistory[36] := 2020, StepHistory[37] := 2030, StepHistory[38] := 9000, StepHistory[39] := 1000, StepHistory[40] := 1010, StepHistory[41] := 1020, StepHistory[42] := 1030, StepHistory[43] := 2000, StepHistory[44] := 2010, StepHistory[45] := 2020, StepHistory[46] := 2030, StepHistory[47] := 2000, StepHistory[48] := 2010, StepHistory[49] := 2020, StepHistory[50] := 2030, StepHistory[51] := 9000, StepHistory[52] := 1000, StepHistory[53] := 1010, StepHistory[54] := 1020, StepHistory[55] := 1030,
        StepHistory[56] := 2000, StepHistory[57] := 2010, StepHistory[58] := 2020, StepHistory[59] := 2030, StepHistory[60] := 2000, StepHistory[61] := 2010, StepHistory[62] := 2020, StepHistory[63] := 2030, AverageCycleTime := 0.060900003, CycleTimeHistory[0] := 0.609, StepTimeHistory[0] := 0.199, StepTimeHistory[2] := 0.2, StepTimeHistory[3] := 0.2, StepTimeHistory[4] := 0.2, StepTimeHistory[7] := 0.199, StepTimeHistory[8] := 0.299, StepTimeHistory[11] := 0.2, StepTimeHistory[12] := 0.298, StepTimeHistory[13] := 0.298, StepTimeHistory[15] := 0.2, StepTimeHistory[16] := 0.298, StepTimeHistory[19] := 0.2, StepTimeHistory[20] := 0.298, StepTimeHistory[23] := 0.2, StepTimeHistory[24] := 4.798, StepTimeHistory[27] := 0.199, StepTimeHistory[28] := 0.199, StepTimeHistory[29] := 0.199, StepTimeHistory[31] := 0.2, StepTimeHistory[32] := 0.2, StepTimeHistory[33] := 0.2, StepTimeHistory[35] := 0.199, StepTimeHistory[36] := 0.199, StepTimeHistory[37] := 0.199, StepTimeHistory[38] := 0.199, StepTimeHistory[40] := 0.199, StepTimeHistory[41] := 0.199, StepTimeHistory[42] := 0.199, StepTimeHistory[44] := 0.2, StepTimeHistory[45] := 0.2, StepTimeHistory[46] := 0.2, StepTimeHistory[48] := 0.199, StepTimeHistory[49] := 0.199, StepTimeHistory[50] := 0.199, StepTimeHistory[51] := 0.199, StepTimeHistory[53] := 0.199, StepTimeHistory[54] := 0.199, StepTimeHistory[55] := 0.199, StepTimeHistory[57] := 0.199, StepTimeHistory[58] := 0.199, StepTimeHistory[59] := 0.199, StepTimeHistory[61] := 0.2, StepTimeHistory[62] := 0.2, StepTimeHistory[63] := 0.2, StepTimer.PRE := 999999999, CycleTimer.PRE := 999999999);
   CTS1_SeqUID : DINT := 9476;
   CTS1_UIDMsg : MESSAGE;
        MessageParameters(ServiceCode := 16#0010, LocalElement := CTS1_Result.UID, ...)
   CTS1_WriteMsg : MESSAGE;
        MessageParameters(ServiceCode := 16#0010, LocalElement := CTS1_BarcodeWrite.DATA[0], ...)
   CTS2_BarcodeWrite : STRING80;
   CTS2_BasicResult : MESSAGE;
        MessageParameters(ServiceCode := 16#000e, DestinationTag := CTS2_Result.Basic, ...)
   CTS2_DataRead : STRING80;
   CTS2_DetailResult : MESSAGE;
        MessageParameters(ServiceCode := 16#000e, DestinationTag := CTS2_Result.Detailed, ...)
   CTS2_Inputs : udt_CTS_INPUTS_FROM := (Discrete_Status_Data := -16384, Active_program_num := 3, unique_id := 10924, channel_num := 1, program_num := 3, sequence_num := 3, seq_unique_ID := 10924, evaluation_code := 1, year := 26, month := 9, date := 28, hour := 11, seconds := 7, flags := 16, test_type := 131, Measurement_data[0].Variable_code := 164, Measurement_data[0].Unit_code := 167, Measurement_data[0].result_measurement := 1.0, Measurement_data[1].Variable_code := 164, Measurement_data[1].Unit_code := 167, Measurement_data[1].result_measurement := 2.0);
   CTS2_LastResultEval : STRING16;
   CTS2_LastTestUID : DINT := 10592;
   CTS2_NextTestUID : DINT := 10592;
   CTS2_NumTestsInSeq : SINT := 2;
   CTS2_Outputs : udt_CTS_OUTPUTS_TO := (program_num := 3);
   CTS2_ReadMsg : MESSAGE;
        MessageParameters(ServiceCode := 16#000e, DestinationTag := CTS2_DataRead.DATA[0], ...)
   CTS2_Ready : DINT;
   CTS2_Result : udt_CTS_RESULT := (UID := 10592, Basic.unique_id := 10592, Basic.channel_num := 1, Basic.program_num := 2, Basic.evaluation_code := 1, Basic.test_port := 1, Basic.year := 26, Basic.month := 9, Basic.date := 25, Basic.hour := 12, Basic.minute := 39, Basic.second := 32, Basic.flags := 12, Basic.Num_tests := 1, Basic.test_elements.test_type := 66, Basic.test_elements.test_eval := 1, Basic.test_elements.num_elements := 16, Detailed.unique_id := 10592, Detailed.num_elements := 16, Detailed.Test_Type := 66, Detailed.element_data[0].Variable_code := 61, Detailed.element_data[0].prec_code := 2, Detailed.element_data[0].Unit_code := 60, Detailed.element_data[0].result_measurement := 0.10728836, Detailed.element_data[1].Variable_code := 28, Detailed.element_data[1].prec_code := 3, Detailed.element_data[1].Unit_code := 41, Detailed.element_data[1].result_measurement := 0.003511086, Detailed.element_data[2].Variable_code := 13, Detailed.element_data[2].prec_code := 3, Detailed.element_data[2].Unit_code := 12, Detailed.element_data[2].result_measurement := 5.0658684, Detailed.element_data[3].Variable_code := 75, Detailed.element_data[3].prec_code := 2, Detailed.element_data[3].Unit_code := 60, Detailed.element_data[4].Variable_code := 60, Detailed.element_data[4].prec_code := 2, Detailed.element_data[4].Unit_code := 60, Detailed.element_data[4].result_measurement := 0.12684613, Detailed.element_data[5].Variable_code := 56, Detailed.element_data[5].prec_code := 3, Detailed.element_data[5].Unit_code := 41, Detailed.element_data[5].result_measurement := 0.0020349398, Detailed.element_data[6].Variable_code := 55, Detailed.element_data[6].prec_code := 3, Detailed.element_data[6].Unit_code := 12, Detailed.element_data[6].result_measurement := 5.0658684, Detailed.element_data[7].Variable_code := 58, Detailed.element_data[7].prec_code := 2, Detailed.element_data[7].Unit_code := 60, Detailed.element_data[7].result_measurement := -1.0002404, Detailed.element_data[8].Variable_code := 59, Detailed.element_data[8].prec_code := 2, Detailed.element_data[8].Unit_code := 60, Detailed.element_data[8].result_measurement := 1.0002404, Detailed.element_data[9].Variable_code := 12, Detailed.element_data[9].prec_code := 3, Detailed.element_data[9].Unit_code := 12, Detailed.element_data[9].result_measurement := 5.000001, Detailed.element_data[10].Variable_code := 62,
        Detailed.element_data[10].prec_code := 2, Detailed.element_data[10].Unit_code := 60, Detailed.element_data[10].result_measurement := 1.0902061, Detailed.element_data[11].Variable_code := 21, Detailed.element_data[11].prec_code := 3, Detailed.element_data[11].Unit_code := 41, Detailed.element_data[11].result_measurement := 0.0015180558, Detailed.element_data[12].Variable_code := 25, Detailed.element_data[12].prec_code := 3, Detailed.element_data[12].Unit_code := 41, Detailed.element_data[12].result_measurement := 0.021727756, Detailed.element_data[13].Variable_code := 216, Detailed.element_data[13].prec_code := 3, Detailed.element_data[13].Unit_code := 41, Detailed.element_data[13].result_measurement := 0.00085681677, Detailed.element_data[14].Variable_code := 218, Detailed.element_data[14].prec_code := 3, Detailed.element_data[14].Unit_code := 41, Detailed.element_data[14].result_measurement := 0.01094304, Detailed.element_data[15].Variable_code := 295, Detailed.element_data[15].prec_code := 3, Detailed.element_data[15].Unit_code := 12, Detailed.element_data[15].result_measurement := 5.0730352);
   CTS2_ResultHistoryLeak : udt_CTS_RESULT[10] := ([0].UID := 10565, [0].Basic.unique_id := 10565, [0].Basic.channel_num := 1, [0].Basic.program_num := 2, [0].Basic.evaluation_code := 1, [0].Basic.test_port := 1, [0].Basic.year := 26, [0].Basic.month := 9, [0].Basic.date := 25, [0].Basic.hour := 12, [0].Basic.minute := 21, [0].Basic.second := 19, [0].Basic.flags := 12, [0].Basic.Num_tests := 1, [0].Basic.test_elements.test_type := 66, [0].Basic.test_elements.test_eval := 1, [0].Basic.test_elements.num_elements := 16, [0].Detailed.unique_id := 10565, [0].Detailed.num_elements := 16, [0].Detailed.Test_Type := 66, [0].Detailed.element_data[0].Variable_code := 61, [0].Detailed.element_data[0].prec_code := 2, [0].Detailed.element_data[0].Unit_code := 60, [0].Detailed.element_data[0].result_measurement := 0.12293458, [0].Detailed.element_data[1].Variable_code := 28, [0].Detailed.element_data[1].prec_code := 3, [0].Detailed.element_data[1].Unit_code := 41, [0].Detailed.element_data[1].result_measurement := 0.003799796, [0].Detailed.element_data[2].Variable_code := 13, [0].Detailed.element_data[2].prec_code := 3, [0].Detailed.element_data[2].Unit_code := 12, [0].Detailed.element_data[2].result_measurement := 5.0659013, [0].Detailed.element_data[3].Variable_code := 75, [0].Detailed.element_data[3].prec_code := 2, [0].Detailed.element_data[3].Unit_code := 60, [0].Detailed.element_data[4].Variable_code := 60, [0].Detailed.element_data[4].prec_code := 2, [0].Detailed.element_data[4].Unit_code := 60, [0].Detailed.element_data[4].result_measurement := 0.1296401, [0].Detailed.element_data[5].Variable_code := 56, [0].Detailed.element_data[5].prec_code := 3, [0].Detailed.element_data[5].Unit_code := 41, [0].Detailed.element_data[5].result_measurement := 0.002058223, [0].Detailed.element_data[6].Variable_code := 55, [0].Detailed.element_data[6].prec_code := 3, [0].Detailed.element_data[6].Unit_code := 12, [0].Detailed.element_data[6].result_measurement := 5.0659013, [0].Detailed.element_data[7].Variable_code := 58, [0].Detailed.element_data[7].prec_code := 2, [0].Detailed.element_data[7].Unit_code := 60, [0].Detailed.element_data[7].result_measurement := -1.0002404, [0].Detailed.element_data[8].Variable_code := 59, [0].Detailed.element_data[8].prec_code := 2, [0].Detailed.element_data[8].Unit_code := 60, [0].Detailed.element_data[8].result_measurement := 1.0002404, [0].Detailed.element_data[9].Variable_code := 12, [0].Detailed.element_data[9].prec_code := 3, [0].Detailed.element_data[9].Unit_code := 12, [0].Detailed.element_data[9].result_measurement := 5.000001, [0].Detailed.element_data[10].Variable_code := 62,
        [0].Detailed.element_data[10].prec_code := 2, [0].Detailed.element_data[10].Unit_code := 60, [0].Detailed.element_data[10].result_measurement := 1.0902061, [0].Detailed.element_data[11].Variable_code := 21, [0].Detailed.element_data[11].prec_code := 3, [0].Detailed.element_data[11].Unit_code := 41, [0].Detailed.element_data[11].result_measurement := 0.0015180558, [0].Detailed.element_data[12].Variable_code := 25, [0].Detailed.element_data[12].prec_code := 3, [0].Detailed.element_data[12].Unit_code := 41, [0].Detailed.element_data[12].result_measurement := 0.021727756, [0].Detailed.element_data[13].Variable_code := 216, [0].Detailed.element_data[13].prec_code := 3, [0].Detailed.element_data[13].Unit_code := 41, [0].Detailed.element_data[13].result_measurement := 0.00085681677, [0].Detailed.element_data[14].Variable_code := 218, [0].Detailed.element_data[14].prec_code := 3, [0].Detailed.element_data[14].Unit_code := 41, [0].Detailed.element_data[14].result_measurement := 0.01094304, [0].Detailed.element_data[15].Variable_code := 295, [0].Detailed.element_data[15].prec_code := 3, [0].Detailed.element_data[15].Unit_code := 12, [0].Detailed.element_data[15].result_measurement := 5.0722575, [1].UID := 10568, [1].Basic.unique_id := 10568, [1].Basic.channel_num := 1, [1].Basic.program_num := 2, [1].Basic.evaluation_code := 1, [1].Basic.test_port := 1, [1].Basic.year := 26, [1].Basic.month := 9, [1].Basic.date := 25, [1].Basic.hour := 12, [1].Basic.minute := 21, [1].Basic.second := 40, [1].Basic.flags := 12, [1].Basic.Num_tests := 1, [1].Basic.test_elements.test_type := 66, [1].Basic.test_elements.test_eval := 1, [1].Basic.test_elements.num_elements := 16, [1].Detailed.unique_id := 10568, [1].Detailed.num_elements := 16, [1].Detailed.Test_Type := 66, [1].Detailed.element_data[0].Variable_code := 61, [1].Detailed.element_data[0].prec_code := 2, [1].Detailed.element_data[0].Unit_code := 60, [1].Detailed.element_data[0].result_measurement := 0.13411045, [1].Detailed.element_data[1].Variable_code := 28, [1].Detailed.element_data[1].prec_code := 3, [1].Detailed.element_data[1].Unit_code := 41, [1].Detailed.element_data[1].result_measurement := 0.0040140003, [1].Detailed.element_data[2].Variable_code := 13, [1].Detailed.element_data[2].prec_code := 3, [1].Detailed.element_data[2].Unit_code := 12, [1].Detailed.element_data[2].result_measurement := 5.0663853, [1].Detailed.element_data[3].Variable_code := 75, [1].Detailed.element_data[3].prec_code := 2, [1].Detailed.element_data[3].Unit_code := 60, [1].Detailed.element_data[4].Variable_code := 60, [1].Detailed.element_data[4].prec_code := 2,
        [1].Detailed.element_data[4].Unit_code := 60, [1].Detailed.element_data[4].result_measurement := 0.12572855, [1].Detailed.element_data[5].Variable_code := 56, [1].Detailed.element_data[5].prec_code := 3, [1].Detailed.element_data[5].Unit_code := 41, [1].Detailed.element_data[5].result_measurement := 0.00202097, [1].Detailed.element_data[6].Variable_code := 55, [1].Detailed.element_data[6].prec_code := 3, [1].Detailed.element_data[6].Unit_code := 12, [1].Detailed.element_data[6].result_measurement := 5.0663853, [1].Detailed.element_data[7].Variable_code := 58, [1].Detailed.element_data[7].prec_code := 2, [1].Detailed.element_data[7].Unit_code := 60, [1].Detailed.element_data[7].result_measurement := -1.0002404, [1].Detailed.element_data[8].Variable_code := 59, [1].Detailed.element_data[8].prec_code := 2, [1].Detailed.element_data[8].Unit_code := 60, [1].Detailed.element_data[8].result_measurement := 1.0002404, [1].Detailed.element_data[9].Variable_code := 12, [1].Detailed.element_data[9].prec_code := 3, [1].Detailed.element_data[9].Unit_code := 12, [1].Detailed.element_data[9].result_measurement := 5.000001, [1].Detailed.element_data[10].Variable_code := 62, [1].Detailed.element_data[10].prec_code := 2, [1].Detailed.element_data[10].Unit_code := 60, [1].Detailed.element_data[10].result_measurement := 1.0902061, [1].Detailed.element_data[11].Variable_code := 21, [1].Detailed.element_data[11].prec_code := 3, [1].Detailed.element_data[11].Unit_code := 41, [1].Detailed.element_data[11].result_measurement := 0.0015180558, [1].Detailed.element_data[12].Variable_code := 25, [1].Detailed.element_data[12].prec_code := 3, [1].Detailed.element_data[12].Unit_code := 41, [1].Detailed.element_data[12].result_measurement := 0.021727756, [1].Detailed.element_data[13].Variable_code := 216, [1].Detailed.element_data[13].prec_code := 3, [1].Detailed.element_data[13].Unit_code := 41, [1].Detailed.element_data[13].result_measurement := 0.00085681677, [1].Detailed.element_data[14].Variable_code := 218, [1].Detailed.element_data[14].prec_code := 3, [1].Detailed.element_data[14].Unit_code := 41, [1].Detailed.element_data[14].result_measurement := 0.01094304, [1].Detailed.element_data[15].Variable_code := 295, [1].Detailed.element_data[15].prec_code := 3, [1].Detailed.element_data[15].Unit_code := 12, [1].Detailed.element_data[15].result_measurement := 5.0729885, [2].UID := 10571, [2].Basic.unique_id := 10571, [2].Basic.channel_num := 1, [2].Basic.program_num := 2, [2].Basic.evaluation_code := 1, [2].Basic.test_port := 1, [2].Basic.year := 26, [2].Basic.month := 9, [2].Basic.date := 25, [2].Basic.hour := 12, [2].Basic.minute := 22, [2].Basic.second := 1, [2].Basic.flags := 12, [2].Basic.Num_tests := 1,
        [2].Basic.test_elements.test_type := 66, [2].Basic.test_elements.test_eval := 1, [2].Basic.test_elements.num_elements := 16, [2].Detailed.unique_id := 10571, [2].Detailed.num_elements := 16, [2].Detailed.Test_Type := 66, [2].Detailed.element_data[0].Variable_code := 61, [2].Detailed.element_data[0].prec_code := 2, [2].Detailed.element_data[0].Unit_code := 60, [2].Detailed.element_data[0].result_measurement := 0.12908131, [2].Detailed.element_data[1].Variable_code := 28, [2].Detailed.element_data[1].prec_code := 3, [2].Detailed.element_data[1].Unit_code := 41, [2].Detailed.element_data[1].result_measurement := 0.003920868, [2].Detailed.element_data[2].Variable_code := 13, [2].Detailed.element_data[2].prec_code := 3, [2].Detailed.element_data[2].Unit_code := 12, [2].Detailed.element_data[2].result_measurement := 5.066935, [2].Detailed.element_data[3].Variable_code := 75, [2].Detailed.element_data[3].prec_code := 2, [2].Detailed.element_data[3].Unit_code := 60, [2].Detailed.element_data[4].Variable_code := 60, [2].Detailed.element_data[4].prec_code := 2, [2].Detailed.element_data[4].Unit_code := 60, [2].Detailed.element_data[4].result_measurement := 0.14137477, [2].Detailed.element_data[5].Variable_code := 56, [2].Detailed.element_data[5].prec_code := 3, [2].Detailed.element_data[5].Unit_code := 41, [2].Detailed.element_data[5].result_measurement := 0.002165325, [2].Detailed.element_data[6].Variable_code := 55, [2].Detailed.element_data[6].prec_code := 3, [2].Detailed.element_data[6].Unit_code := 12, [2].Detailed.element_data[6].result_measurement := 5.066935, [2].Detailed.element_data[7].Variable_code := 58, [2].Detailed.element_data[7].prec_code := 2, [2].Detailed.element_data[7].Unit_code := 60, [2].Detailed.element_data[7].result_measurement := -1.0002404, [2].Detailed.element_data[8].Variable_code := 59, [2].Detailed.element_data[8].prec_code := 2, [2].Detailed.element_data[8].Unit_code := 60, [2].Detailed.element_data[8].result_measurement := 1.0002404, [2].Detailed.element_data[9].Variable_code := 12, [2].Detailed.element_data[9].prec_code := 3, [2].Detailed.element_data[9].Unit_code := 12, [2].Detailed.element_data[9].result_measurement := 5.000001, [2].Detailed.element_data[10].Variable_code := 62, [2].Detailed.element_data[10].prec_code := 2, [2].Detailed.element_data[10].Unit_code := 60, [2].Detailed.element_data[10].result_measurement := 1.0902061, [2].Detailed.element_data[11].Variable_code := 21, [2].Detailed.element_data[11].prec_code := 3, [2].Detailed.element_data[11].Unit_code := 41, [2].Detailed.element_data[11].result_measurement := 0.0015180558, [2].Detailed.element_data[12].Variable_code := 25, [2].Detailed.element_data[12].prec_code := 3, [2].Detailed.element_data[12].Unit_code := 41, [2].Detailed.element_data[12].result_measurement := 0.021727756, [2].Detailed.element_data[13].Variable_code := 216, [2].Detailed.element_data[13].prec_code := 3, [2].Detailed.element_data[13].Unit_code := 41,
